# B&R Automation Studio project TD52 (part 79)

#### fPCGVmon.c
```c
/********************************************************************
 * COPYRIGHT -- B&R Industrial Automation GmbH
 ********************************************************************
 * Program: PCGVmon
 * File: fPCGVmon.c
 * Author: 105055527
 * Last modified by: schmisi00
 * Created: Mon Sep 05 18:14:57 2016
 * Last modified: Thu Nov 26 09:45:08 2020
 * Model Version: 0.03
 * Description: Pre-chamber gas valve monitoring (sticking detection).

   Outstandings:
   -------------
   - NA
 * modified Comment: V0.01    22.09.2020    Schmidt,   created initial model
   V0.02    15.10.2020    Schmidt,   modifications after code review / unit testing
   V0.03    26.11.2020    Schmidt,   perm's for class borders (no-hardcoded borders)
 ********************************************************************
 * Implementation of program PCGVmon
 ********************************************************************
 * Generated with B&R Automation Studio Target for Simulink V6.2.0
 * (ERT based)
 ********************************************************************/

#include <bur/plctypes.h>
#include "PCGVmon.h"
#include "rtwtypes.h"

/* Defines */
#define SS_TERMINATE 4
#define SS_OUTPUT 3
#define SS_INITIALIZE 2

/*  Data Types */

/**************************** GLOBAL DATA *************************************/
/*  Definitions */

/*  Declarations  */

/***************************** FILE SCOPE DATA ********************************/

/*************************** FUNCTIONS ****************************************/
#ifdef __cplusplus

unsigned long bur_heap_size = 6553500;

#endif

/*LEGACYMODE_VARIABLES*/
void fPCGVmon(struct fPCGVmon* inst)
{
  tag_RTM_PCGVmon* const PCGVmon_M = &(inst)->bur_PCGVmon;
	inst->bur_PCGVmon.blockIO = &(inst)->bur_BlockIO_PCGVmon;
	inst->bur_PCGVmon.inputs = &(inst)->bur_ExternalInputs_PCGVmon;
	inst->bur_PCGVmon.outputs = &(inst)->bur_ExternalOutputs_PCGVmon;
	inst->bur_PCGVmon.dwork = &(inst)->bur_D_Work_PCGVmon;

  switch (inst->ssMethodType)
  {
   case SS_INITIALIZE:
    /* call model initialize function */
    PCGVmon_initialize(PCGVmon_M, inst);
    break;

   case SS_OUTPUT:
    /* call model step function */
    PCGVmon_step(PCGVmon_M, inst);

    break;

   case SS_TERMINATE:
    /* call model terminate function */
    PCGVmon_terminate(PCGVmon_M, inst);
    break;
  }
}

/*****************************************************************************
   Function block sample time: 1.0s
 *****************************************************************************/

/*****************************************************************************
   B&R Automation Studio Target for Simulink Version: A6.2.0 (28-May-2020)
 *****************************************************************************/

/*======================== TOOL VERSION INFORMATION ==========================*
 * MATLAB 9.8 (R2020a)18-Nov-2019                                             *
 * Simulink 10.1 (R2020a)18-Nov-2019                                          *
 * Simulink Coder 9.3 (R2020a)18-Nov-2019                                     *
 * Embedded Coder 7.4 (R2020a)18-Nov-2019                                     *
 * Stateflow 10.2 (R2020a)18-Nov-2019                                         *
 *============================================================================*/

/*======================= LICENSE IN USE INFORMATION =========================*
 * matlab                                                                     *
 * matlab_coder                                                               *
 * real-time_workshop                                                         *
 * rtw_embedded_coder                                                         *
 * simulink                                                                   *
 *============================================================================*/
```

#### lPCGVmon.fun
```iecst
FUNCTION_BLOCK fPCGVmon
  VAR_INPUT
    ssMethodType: SINT;
  END_VAR
  VAR_INPUT
        Input : tPCGVmon_IN; (*PCGV monitoring bus inputs*)
  END_VAR
  VAR_INPUT
        Perm : tPCGVmon_PERM; (*PCGV monitoring bus perms*)
  END_VAR
  VAR_OUTPUT
        Debug : tPCGVmon_DBG; (*PCGV monitoring bus debug*)
  END_VAR
  VAR_OUTPUT
        Output : tPCGVmon_OUT; (*PCGV monitoring bus outputs*)
  END_VAR
  VAR_OUTPUT
        Version : UDINT; (**)
  END_VAR
	VAR
		bur_BlockIO_PCGVmon : BlockIO_PCGVmon;
	END_VAR
	VAR
		bur_ExternalInputs_PCGVmon : ExternalInputs_PCGVmon;
	END_VAR
	VAR
		bur_ExternalOutputs_PCGVmon : ExternalOutputs_PCGVmon;
	END_VAR
	VAR
		bur_D_Work_PCGVmon : D_Work_PCGVmon;
	END_VAR
	VAR
		bur_PCGVmon : tag_RTM_PCGVmon;
	END_VAR
END_FUNCTION_BLOCK
```

#### lPCGVmon.typ
```iecst
TYPE
	tPCGVmon_DBG :  STRUCT
		bPCGVstick :  ARRAY[0..24] OF BOOL; (*PCGVstickingevent(-)*)
		rTexh_median_diff_grad :  ARRAY[0..24] OF REAL; (**)
		rStdDev :  REAL; (**)
		detectionLim :  REAL; (**)
		rTexh_median_filt :  REAL; (**)
		rU_Ign_Act_Filt :  ARRAY[0..24] OF REAL; (**)
		rTexhMedDeviat :  ARRAY[0..24] OF REAL; (**)
		count1_stick :  ARRAY[0..24] OF REAL; (**)
		count2_stickLong :  ARRAY[0..24] OF REAL; (**)
		unstickDet :  ARRAY[0..24] OF REAL; (**)
		multStickDur :  ARRAY[0..24] OF REAL; (**)
		tiStickDurAll :  ARRAY[0..24] OF REAL; (**)
		bPCGVstickALL :  ARRAY[0..24] OF BOOL; (*PCGVstickingevent(-)*)
		bTexhInRange_out :  ARRAY[0..24] OF BOOL; (*EGTwithinlimit/range(-)*)
	END_STRUCT;

	tPCGVmon_IN :  STRUCT
		rU_Ign_Act :  ARRAY[0..24] OF REAL; (*Actualcylinderignitionvoltage(kV)*)
		MSAGT :  ARRAY[0..24] OF BOOL; (*Cylinderexhaustgastemperaturesensorfailure(-)*)
		rT_EPU_EG :  ARRAY[0..24] OF REAL; (*Cylinderexhaustgastemperature(°C)*)
		tGCB_On_Di :  BOOL; (*Generatorcircuitbreakerclosed(-)*)
		ucNumCyl :  USINT; (*Totalnumberofcylinders(-)*)
		iCnt_PCGV_class1_MM2VIS :  ARRAY[0..24] OF UINT; (*Permclass1counter(MM2VIS)*)
		iCnt_PCGV_class2_MM2VIS :  ARRAY[0..24] OF UINT; (*Permclass2counter(MM2VIS)*)
		iCnt_PCGV_class3_MM2VIS :  ARRAY[0..24] OF UINT; (*Permclass3counter(MM2VIS)*)
		iCnt_PCGV_class4_MM2VIS :  ARRAY[0..24] OF UINT; (*Permclass4counter(MM2VIS)*)
	END_STRUCT;

	tPCGVmon_OUT :  STRUCT
		iCnt_PCGV_class1 :  ARRAY[0..24] OF UINT; (*Class1counter:stickingduration1-10s*)
		iCnt_PCGV_class2 :  ARRAY[0..24] OF UINT; (*Class2counter:stickingduration10-60s*)
		iCnt_PCGV_class3 :  ARRAY[0..24] OF UINT; (*Class3counter:stickingduration60-300s*)
		iCnt_PCGV_class4 :  ARRAY[0..24] OF UINT; (*Class3counter:stickingduration300-3600s*)
		rTi_PCGV_LastStickDur :  REAL; (*Laststickingduration(s)*)
		rTi_PCGV_MeanLastStickEvts :  REAL; (*Stickingdurationoflaststickingevents(s)*)
	END_STRUCT;

	tPCGVmon_PERM :  STRUCT
		bPCGVmon_Act :  BOOL; (*ActivationofPCGVmonitoringandclasscoutnerreset(-)*)
		rU_Ign_DetLim :  REAL; (*MaximumignitionvoltagedroptostillconsiderEGTtemperaturedropasPCGVsticking(kV)*)
		rU_Ign_CylActThresh :  REAL; (*CylinderEGTbelowthisparametertimesignitionvoltagemedianexcludedfrommonitoring(-)*)
		rT_recoverLim :  REAL; (*CylinderEGTrecoverthreshold(°C)*)
		rTi_Uign_MonActDelay :  REAL; (*Activationdelayforignitionvoltageconsiderationinmonitoringfunction(s)*)
		rTmedian_StartThresh :  REAL; (*EGT(median)tobereachedforactivationofignitionvoltageconsideration(°C)*)
		rTi_GCBon_Delay :  REAL; (*ActivationdelayafterGCBclosed(s)*)
		rTi_EGT_ss_ActDelay :  REAL; (*ActivationdelayafterEGTissteadystate(s)*)
		rOffset_EGTgradient_trans :  REAL; (*EGTgradientdetectionlimitoffsetfortransients(-)*)
		rOffset_EGTgradient_ss :  REAL; (*EGTgradientdetectionlimitoffsetforsteadystate(-)*)
		rGradient_LimSwitch :  REAL; (*Switchdetectionlimit(-)*)
		iCnt_PCGV_class1 :  ARRAY[0..24] OF UINT; (*Permclass1counter:stickingduration1-10s*)
		iCnt_PCGV_class2 :  ARRAY[0..24] OF UINT; (*Permclass2counter:stickingduration10-60s*)
		iCnt_PCGV_class3 :  ARRAY[0..24] OF UINT; (*Permclass3counter:stickingduration60-300s*)
		iCnt_PCGV_class4 :  ARRAY[0..24] OF UINT; (*Permclass4counter:stickingduration300-3600s*)
		iTi_PCGV_class1_border :  UINT; (*Permclass1border*)
		iTi_PCGV_class2_border :  UINT; (*Permclass2border*)
		iTi_PCGV_class3_border :  UINT; (*Permclass3border*)
		iTi_PCGV_class4_border :  UINT; (*Permclass4border*)
	END_STRUCT;

END_TYPE

TYPE
rtB_setZero_PCGVmon : STRUCT
	y : ARRAY[0..24] OF REAL;
END_STRUCT;
rtB_TON_PCGVmon : STRUCT
	LogicalOperator3 : BOOL;
END_STRUCT;
rtDW_TON_PCGVmon : STRUCT
	DiscreteTimeIntegrator_DSTATE : REAL;
	DiscreteTimeIntegrator_PrevRese : SINT;
END_STRUCT;
rtB_MATLABFunction_PCGVmon : STRUCT
	y : REAL;
END_STRUCT;
BlockIO_PCGVmon : STRUCT
	BusConversion_InsertedFor_BusOu : tPCGVmon_DBG;
	BusInput : tPCGVmon_IN;
	BusInput1 : tPCGVmon_PERM;
	BusConversion_InsertedFor_Bus_d : tPCGVmon_OUT;
	UnitDelay : UDINT;
	sf_MATLABFunction9 : rtB_MATLABFunction_PCGVmon;
	sf_MATLABFunction8 : rtB_MATLABFunction_PCGVmon;
	sf_MATLABFunction7 : rtB_MATLABFunction_PCGVmon;
	sf_MATLABFunction6 : rtB_MATLABFunction_PCGVmon;
	sf_MATLABFunction5 : rtB_MATLABFunction_PCGVmon;
	sf_MATLABFunction4 : rtB_MATLABFunction_PCGVmon;
	sf_MATLABFunction3_o : rtB_MATLABFunction_PCGVmon;
	sf_MATLABFunction2_o : rtB_MATLABFunction_PCGVmon;
	sf_MATLABFunction10 : rtB_MATLABFunction_PCGVmon;
	sf_MATLABFunction1_p : rtB_MATLABFunction_PCGVmon;
	sf_MATLABFunction : rtB_MATLABFunction_PCGVmon;
	sf_setZero_m : rtB_setZero_PCGVmon;
	TON2 : rtB_TON_PCGVmon;
	TON1 : rtB_TON_PCGVmon;
	TON : rtB_TON_PCGVmon;
	sf_setZero1 : rtB_setZero_PCGVmon;
	sf_setZero : rtB_setZero_PCGVmon;
END_STRUCT;
D_Work_PCGVmon : STRUCT
	Delay_DSTATE : ARRAY[0..74] OF REAL;
	Delay1_DSTATE : ARRAY[0..24] OF REAL;
	UnitDelay2_DSTATE : ARRAY[0..24] OF REAL;
	DelayInput1_DSTATE : REAL;
	UnitDelay13_DSTATE : REAL;
	UnitDelay3_DSTATE : REAL;
	UnitDelay4_DSTATE : REAL;
	UnitDelay5_DSTATE : REAL;
	UnitDelay6_DSTATE : REAL;
	UnitDelay7_DSTATE : REAL;
	UnitDelay8_DSTATE : REAL;
	UnitDelay9_DSTATE : REAL;
	UnitDelay10_DSTATE : REAL;
	UnitDelay11_DSTATE : REAL;
	UnitDelay12_DSTATE : REAL;
	DiscreteTimeIntegrator_DSTATE : REAL;
	DiscreteTimeIntegrator_DSTATE_d : ARRAY[0..24] OF REAL;
	DiscreteTimeIntegrator_DSTATE_b : REAL;
	DiscreteTimeIntegrator_DSTATE_m : ARRAY[0..24] OF REAL;
	UnitDelay_DSTATE : UDINT;
	PrevY : REAL;
	PrevY_a : REAL;
	Cnt1OldDely : ARRAY[0..24] OF REAL;
	Cnt2Old : ARRAY[0..24] OF REAL;
	lastStickDurTmp : ARRAY[0..24] OF REAL;
	count1 : ARRAY[0..24] OF REAL;
	count2 : ARRAY[0..24] OF REAL;
	tiStickDur : ARRAY[0..24] OF REAL;
	tiMultStick : ARRAY[0..24] OF REAL;
	tiStickDurAll : ARRAY[0..24] OF REAL;
	count1Old : ARRAY[0..24] OF REAL;
	iCnt_class1 : ARRAY[0..24] OF UINT;
	iCnt_class2 : ARRAY[0..24] OF UINT;
	iCnt_class3 : ARRAY[0..24] OF UINT;
	iCnt_class4 : ARRAY[0..24] OF UINT;
	iCnt_class1Old : ARRAY[0..24] OF UINT;
	iCnt_class2Old : ARRAY[0..24] OF UINT;
	iCnt_class3Old : ARRAY[0..24] OF UINT;
	iCnt_class4Old : ARRAY[0..24] OF UINT;
	DiscreteTimeIntegrator_PrevRese : SINT;
	DiscreteTimeIntegrator_PrevRe_a : SINT;
	DiscreteTimeIntegrator_PrevRe_p : SINT;
	DiscreteTimeIntegrator_PrevRe_l : SINT;
	DiscreteTimeIntegrator_IC_LOADI : USINT;
	DiscreteTimeIntegrator_IC_LOA_b : USINT;
	DiscreteTimeIntegrator_IC_LOA_l : USINT;
	DiscreteTimeIntegrator_IC_LOA_o : USINT;
	Relay1_Mode : ARRAY[0..24] OF BOOL;
	bPCGVstickTexhGradOld : ARRAY[0..24] OF BOOL;
	bPCGVstick_temp : ARRAY[0..24] OF BOOL;
	bPCGVstickOld : ARRAY[0..24] OF BOOL;
	switch1 : ARRAY[0..24] OF BOOL;
	switch2 : ARRAY[0..24] OF BOOL;
	switch3 : ARRAY[0..24] OF BOOL;
	bTexhInRangeOld : ARRAY[0..24] OF BOOL;
	bTexhInRange : ARRAY[0..24] OF BOOL;
	GCBold : BOOL;
	TON2 : rtDW_TON_PCGVmon;
	TON1 : rtDW_TON_PCGVmon;
	TON : rtDW_TON_PCGVmon;
END_STRUCT;
ExternalInputs_PCGVmon : STRUCT
	In : tPCGVmon_IN;
	Perm : tPCGVmon_PERM;
END_STRUCT;
ExternalOutputs_PCGVmon : STRUCT
	Out : tPCGVmon_OUT;
	Dbg : tPCGVmon_DBG;
END_STRUCT;
tag_RTM_PCGVmon : STRUCT
	errorStatus : REFERENCE TO USINT;
	blockIO : REFERENCE TO BlockIO_PCGVmon;
	inputs : REFERENCE TO ExternalInputs_PCGVmon;
	outputs : REFERENCE TO ExternalOutputs_PCGVmon;
	dwork : REFERENCE TO D_Work_PCGVmon;
END_STRUCT;
emxArray_int32_T_25_PCGVmon : emxArray_int32_T_25;

RT_MODEL_PCGVmon : tag_RTM_PCGVmon;

END_TYPE
TYPE
emxArray_int32_T_25 : STRUCT
	data : ARRAY[0..24] OF DINT;
	size : DINT;
END_STRUCT;
END_TYPE
```

#### lib_properties.txt
```
For manual assignment to hardware configuration please
add the following additional include directories:

\Logical\MATLAB_includes\R2020a\

And the following additional build options:

-lm -D MODEL=PCGVmon -D NUMST=1 -D NCSTATES=0 -D HAVESTDIO -D MODEL_HAS_DYNAMICALLY_LOADED_SFCNS=0 -D CLASSIC_INTERFACE=0 -D ALLOCATIONFCN=0 -D TID01EQ=0 -D TERMFCN=1 -D ONESTEPFCN=1 -D MAT_FILE=0 -D MULTI_INSTANCE_CODE=1 -D INTEGER_CODE=0 -D MT=0
```

#### rt_defines.h
```c
/********************************************************************
 * COPYRIGHT -- B&R Industrial Automation GmbH
 ********************************************************************
 * Program: PCGVmon
 * File: rt_defines.h
 * Author: 105055527
 * Last modified by: schmisi00
 * Created: Mon Sep 05 18:14:57 2016
 * Last modified: Thu Nov 26 09:45:08 2020
 * Model Version: 0.03
 * Description: Pre-chamber gas valve monitoring (sticking detection).

   Outstandings:
   -------------
   - NA
 * modified Comment: V0.01    22.09.2020    Schmidt,   created initial model
   V0.02    15.10.2020    Schmidt,   modifications after code review / unit testing
   V0.03    26.11.2020    Schmidt,   perm's for class borders (no-hardcoded borders)
 ********************************************************************
 * Header for program PCGVmon
 ********************************************************************
 * Generated with B&R Automation Studio Target for Simulink V6.2.0
 * (ERT based)
 ********************************************************************/

#ifndef RTW_HEADER_rt_defines_h_
#define RTW_HEADER_rt_defines_h_
#ifndef MIN
#define MIN(a,b)                       ((a) < (b) ? (a) : (b))
#endif

#ifndef MAX
#define MAX(a,b)                       ((a) > (b) ? (a) : (b))
#endif

#ifndef AST_ROUND
#define AST_ROUND(x)                   ((x)>=0?(long long)((x)+0.5):(long long)((x)-0.5))
#endif

/*===========*
 * Constants *
 *===========*/
#define RT_PI                          3.14159265358979323846
#define RT_PIF                         3.1415927F
#define RT_LN_10                       2.30258509299404568402
#define RT_LN_10F                      2.3025851F
#define RT_LOG10E                      0.43429448190325182765
#define RT_LOG10EF                     0.43429449F
#define RT_E                           2.7182818284590452354
#define RT_EF                          2.7182817F

/*
 * UNUSED_PARAMETER(x)
 *   Used to specify that a function parameter (argument) is required but not
 *   accessed by the function body.
 */
#ifndef UNUSED_PARAMETER
# if defined(__LCC__)
#   define UNUSED_PARAMETER(x)                                   /* do nothing */
# else

/*
 * This is the semi-ANSI standard way of indicating that an
 * unused function parameter is required.
 */
#   define UNUSED_PARAMETER(x)         (void) (x)
# endif
#endif
#endif                                 /* RTW_HEADER_rt_defines_h_ */
```

#### rtwtypes.h
```c
/********************************************************************
 * COPYRIGHT -- B&R Industrial Automation GmbH
 ********************************************************************
 * Program: PCGVmon
 * File: rtwtypes.h
 * Author: 105055527
 * Last modified by: schmisi00
 * Created: Mon Sep 05 18:14:57 2016
 * Last modified: Thu Nov 26 09:45:08 2020
 * Model Version: 0.03
 * Description: Pre-chamber gas valve monitoring (sticking detection).

   Outstandings:
   -------------
   - NA
 * modified Comment: V0.01    22.09.2020    Schmidt,   created initial model
   V0.02    15.10.2020    Schmidt,   modifications after code review / unit testing
   V0.03    26.11.2020    Schmidt,   perm's for class borders (no-hardcoded borders)
 ********************************************************************
 * Header for program PCGVmon
 ********************************************************************
 * Generated with B&R Automation Studio Target for Simulink V6.2.0
 * (ERT based)
 ********************************************************************/

#ifndef RTWTYPES_H
#define RTWTYPES_H

/* Logical type definitions */
#if (!defined(__cplusplus))
#  ifndef false
#   define false                       (0U)
#  endif

#  ifndef true
#   define true                        (1U)
#  endif
#endif

/*=======================================================================*
 * Target hardware information
 *   Device type: Intel->x86/Pentium
 *   Number of bits:     char:   8    short:   16    long:  32
 *                       long:  32
 *                       native word size:  32
 *   Byte ordering: LittleEndian
 *   Signed integer division rounds to: Zero
 *   Shift right on a signed integer as arithmetic shift: on
 *=======================================================================*/

/*=======================================================================*
 * Fixed width word size data types:                                     *
 *   int8_T, int16_T, int32_T     - signed 8, 16, or 32 bit integers     *
 *   uint8_T, uint16_T, uint32_T  - unsigned 8, 16, or 32 bit integers   *
 *   real32_T, real64_T           - 32 and 64 bit floating point numbers *
 *=======================================================================*/
typedef signed char int8_T;
typedef unsigned char uint8_T;
typedef short int16_T;
typedef unsigned short uint16_T;
typedef long int32_T;
typedef unsigned long uint32_T;
typedef float real32_T;
typedef double real64_T;

/*===========================================================================*
 * Generic type definitions: boolean_T, char_T, byte_T, int_T, uint_T,       *
 *                           real_T, time_T, ulong_T.                        *
 *===========================================================================*/
typedef double real_T;
typedef double time_T;
typedef unsigned char boolean_T;
typedef long int_T;
typedef unsigned long uint_T;
typedef unsigned long ulong_T;
typedef char char_T;
typedef unsigned char uchar_T;
typedef char_T byte_T;

/*=======================================================================*
 * Min and Max:                                                          *
 *   int8_T, int16_T, int32_T     - signed 8, 16, or 32 bit integers     *
 *   uint8_T, uint16_T, uint32_T  - unsigned 8, 16, or 32 bit integers   *
 *=======================================================================*/
#define MAX_int8_T                     ((int8_T)(127))
#define MIN_int8_T                     ((int8_T)(-128))
#define MAX_uint8_T                    ((uint8_T)(255U))
#define MAX_int16_T                    ((int16_T)(32767))
#define MIN_int16_T                    ((int16_T)(-32768))
#define MAX_uint16_T                   ((uint16_T)(65535U))
#define MAX_int32_T                    ((int32_T)(2147483647))
#define MIN_int32_T                    ((int32_T)(-2147483647-1))
#define MAX_uint32_T                   ((uint32_T)(0xFFFFFFFFU))

/* Block D-Work pointer type */
typedef void * pointer_T;

#endif                                 /* RTWTYPES_H */

#ifndef MIN
#define MIN(a,b)                       ((a) < (b) ? (a) : (b))
#endif

#ifndef MAX
#define MAX(a,b)                       ((a) > (b) ? (a) : (b))
#endif

#ifndef AST_ROUND
#define AST_ROUND(x)                   ((x)>=0?(long long)((x)+0.5):(long long)((x)-0.5))
#endif
```

### Library Logical/EngineController/Lib_EC/lFSyPrM (ANSIC, version 1.00.0)

#### FSyPrM.c
```c
/********************************************************************
 * COPYRIGHT -- B&R Industrial Automation GmbH
 ********************************************************************
 * Program: FSyPrM
 * File: FSyPrM.c
 * Author: 105055527
 * Last modified by: schmisi00
 * Created: Mon Sep 05 18:14:57 2016
 * Last modified: Mon Jan 25 17:32:20 2021
 * Model Version: 0.08
 * Description: Fast synchronization controller for pre-mixed engines.

   Outstandings:
   -------------
   - NA
 * modified Comment: V0.01    30.03.2020    Schmidt,   project/controller carryover from FSync to FSyncPrM
   V0.02    02.04.2020    Schmidt,   cleanup and deletion of functions not used by pre-mixed engines
   V0.03    12.05.2020    Schmidt,   upgrade to MATLAB/SIMULINK R2020a
   V0.04    14.05.2020    Schmidt,   B&R blocks upgrade to AS Target v6.2.0 (officially supports MATLAB 2020a)
   V0.05    03.08.2020    Schmidt,   changed speed reference for function activation from nominal speed (parameter) to bus bar frequency
   added detection for speed exceedance --> switch over to standard idle controller
   V0.06    04.08.2020    Schmidt,   moved function activation from PARA bus to IN bus
   V0.07    17.08.2020    Schmidt,   included modifications after P6 tests
   V0.08    25.01.2021    Schmidt,   use of frequency based speed set-point (rN_Set) only if rF_MMD_BusBar > 0.5*rF_Nom
 ********************************************************************
 * Implementation of program FSyPrM
 ********************************************************************
 * Generated with B&R Automation Studio Target for Simulink V6.3.1
 * (ERT based)
 ********************************************************************/

#include "FSyPrM.h"
#include "FSyPrM_private.h"

/*  Defines */

/*  Data Types */

/**************************** GLOBAL DATA *************************************/
/*  Definitions */

/*  Declarations  */

/***************************** FILE SCOPE DATA ********************************/

/*************************** FUNCTIONS ****************************************/

/* Model step function */
void FSyPrM_step(RT_MODEL_FSyPrM *const FSyPrM_M, struct fFSyPrM* inst)
{
  struct BlockIO_FSyPrM *FSyPrM_B = ((struct BlockIO_FSyPrM *) FSyPrM_M->blockIO);
  struct D_Work_FSyPrM *FSyPrM_DWork = ((struct D_Work_FSyPrM *) FSyPrM_M->dwork);
  ExternalOutputs_FSyPrM *FSyPrM_Y = (ExternalOutputs_FSyPrM *)
    FSyPrM_M->outputs;
  boolean_T bEnabled;
  real32_T rN_err;
  real32_T rAngle_err;
  real32_T S;
  real32_T gk;
  boolean_T Sf1;
  boolean_T Sf2;
  boolean_T Gplus;
  boolean_T Gminus;
  boolean_T Gammaplus;
  boolean_T Gammaminus;
  boolean_T H1;
  boolean_T H3;
  real32_T rtb_Switch1_i;
  real32_T rtb_DiscreteTimeIntegrator_g;
  int8_T rtb_Switch2;
  real_T rtb_Switch1;
  real32_T S_tmp;
  uint32_T tmp;
  real32_T tmp_0;

  /* S-Function (bur_bus_in): '<Root>/Bus Input' */
  FSyPrM_B->BusInput = inst->In;

  /* S-Function (bur_bus_in): '<Root>/Bus Input1' */
  FSyPrM_B->BusInput1 = inst->Para;

  /* S-Function (bur_bus_in): '<Root>/Bus Input2' */
  FSyPrM_B->BusInput2 = inst->Perm;

  /* Switch: '<S9>/Switch1' incorporates:
   *  Product: '<S9>/Divide1'
   *  Switch: '<S2>/Environment Switch'
   *  Switch: '<S3>/Environment Switch'
   *  Switch: '<S4>/Environment Switch'
   */
  if (FSyPrM_B->BusInput2.bF_act_ena) {
    /* Switch: '<S16>/Switch' incorporates:
     *  Abs: '<S16>/Abs'
     *  RelationalOperator: '<S16>/Relational Operator'
     *  Switch: '<S4>/Environment Switch'
     */
    if (1.0F >= (real32_T)fabs(FSyPrM_B->BusInput1.rF_Nom)) {
      gk = 1.0F;
    } else {
      gk = FSyPrM_B->BusInput1.rF_Nom;
    }

    /* End of Switch: '<S16>/Switch' */
    rtb_Switch1_i = FSyPrM_B->BusInput.rF_MMD * FSyPrM_B->BusInput1.rN_EngNom /
      gk;
  } else {
    rtb_Switch1_i = FSyPrM_B->BusInput.rN_Eng;
  }

  /* End of Switch: '<S9>/Switch1' */

  /* Outputs for Atomic SubSystem: '<S1>/Filter' */
  /* DiscreteIntegrator: '<S10>/Discrete-Time Integrator' incorporates:
   *  Switch: '<S2>/Environment Switch'
   */
  if (FSyPrM_DWork->DiscreteTimeIntegrator_IC_LO_dn != 0) {
    FSyPrM_DWork->DiscreteTimeIntegrator_DSTATE_k = rtb_Switch1_i;
  }

  if (FSyPrM_B->BusInput.bReset ||
      (FSyPrM_DWork->DiscreteTimeIntegrator_PrevRe_d != 0)) {
    FSyPrM_DWork->DiscreteTimeIntegrator_DSTATE_k = rtb_Switch1_i;
  }

  rtb_DiscreteTimeIntegrator_g = FSyPrM_DWork->DiscreteTimeIntegrator_DSTATE_k;

  /* Update for DiscreteIntegrator: '<S10>/Discrete-Time Integrator' */
  FSyPrM_DWork->DiscreteTimeIntegrator_IC_LO_dn = 0U;

  /* Switch: '<S12>/Switch' incorporates:
   *  Abs: '<S12>/Abs'
   *  RelationalOperator: '<S12>/Relational Operator'
   *  Switch: '<S3>/Environment Switch'
   */
  if (2.22044605E-16F >= (real32_T)fabs(FSyPrM_B->BusInput2.rTi_Filtn)) {
    gk = 2.22044605E-16F;
  } else {
    gk = FSyPrM_B->BusInput2.rTi_Filtn;
  }

  /* End of Switch: '<S12>/Switch' */

  /* Update for DiscreteIntegrator: '<S10>/Discrete-Time Integrator' incorporates:
   *  Product: '<S10>/Divide4'
   *  Sum: '<S10>/Sum4'
   *  Switch: '<S2>/Environment Switch'
   */
  FSyPrM_DWork->DiscreteTimeIntegrator_DSTATE_k += (rtb_Switch1_i -
    FSyPrM_DWork->DiscreteTimeIntegrator_DSTATE_k) / gk * 0.01F;
  FSyPrM_DWork->DiscreteTimeIntegrator_PrevRe_d = (int8_T)
    FSyPrM_B->BusInput.bReset;

  /* End of Outputs for SubSystem: '<S1>/Filter' */

  /* Outputs for Atomic SubSystem: '<S1>/Filter1' */
  /* DiscreteIntegrator: '<S11>/Discrete-Time Integrator' incorporates:
   *  Switch: '<S2>/Environment Switch'
   */
  if (FSyPrM_DWork->DiscreteTimeIntegrator_IC_LOA_d != 0) {
    FSyPrM_DWork->DiscreteTimeIntegrator_DSTATE_g = rtb_DiscreteTimeIntegrator_g;
  }

  if (FSyPrM_B->BusInput.bReset ||
      (FSyPrM_DWork->DiscreteTimeIntegrator_PrevRe_h != 0)) {
    FSyPrM_DWork->DiscreteTimeIntegrator_DSTATE_g = rtb_DiscreteTimeIntegrator_g;
  }

  /* Product: '<S11>/Divide4' incorporates:
   *  DiscreteIntegrator: '<S11>/Discrete-Time Integrator'
   *  Sum: '<S11>/Sum4'
   */
  rtb_DiscreteTimeIntegrator_g = (rtb_DiscreteTimeIntegrator_g -
    FSyPrM_DWork->DiscreteTimeIntegrator_DSTATE_g) / 0.01F;

  /* Switch: '<S11>/Switch1' incorporates:
   *  Constant: '<S11>/Constant'
   *  Switch: '<S2>/Environment Switch'
   */
  if (FSyPrM_B->BusInput.bReset) {
    rtb_Switch1 = 0.0;
  } else {
    rtb_Switch1 = rtb_DiscreteTimeIntegrator_g;
  }

  /* End of Switch: '<S11>/Switch1' */

  /* Update for DiscreteIntegrator: '<S11>/Discrete-Time Integrator' incorporates:
   *  Switch: '<S2>/Environment Switch'
   */
  FSyPrM_DWork->DiscreteTimeIntegrator_IC_LOA_d = 0U;
  FSyPrM_DWork->DiscreteTimeIntegrator_DSTATE_g += 0.01F *
    rtb_DiscreteTimeIntegrator_g;
  FSyPrM_DWork->DiscreteTimeIntegrator_PrevRe_h = (int8_T)
    FSyPrM_B->BusInput.bReset;

  /* End of Outputs for SubSystem: '<S1>/Filter1' */

  /* Outputs for Atomic SubSystem: '<S9>/Filter' */
  /* DiscreteIntegrator: '<S18>/Discrete-Time Integrator' incorporates:
   *  Switch: '<S2>/Environment Switch'
   *  Switch: '<S4>/Environment Switch'
   */
  if (FSyPrM_DWork->DiscreteTimeIntegrator_IC_LOADI != 0) {
    FSyPrM_DWork->DiscreteTimeIntegrator_DSTATE = FSyPrM_B->BusInput1.rN_EngNom;
  }

  if (FSyPrM_B->BusInput.bReset ||
      (FSyPrM_DWork->DiscreteTimeIntegrator_PrevRese != 0)) {
    FSyPrM_DWork->DiscreteTimeIntegrator_DSTATE = FSyPrM_B->BusInput1.rN_EngNom;
  }

  rtb_DiscreteTimeIntegrator_g = FSyPrM_DWork->DiscreteTimeIntegrator_DSTATE;

  /* Update for DiscreteIntegrator: '<S18>/Discrete-Time Integrator' */
  FSyPrM_DWork->DiscreteTimeIntegrator_IC_LOADI = 0U;

  /* End of Outputs for SubSystem: '<S9>/Filter' */

  /* Switch: '<S17>/Switch' incorporates:
   *  Abs: '<S17>/Abs'
   *  RelationalOperator: '<S17>/Relational Operator'
   *  Switch: '<S4>/Environment Switch'
   */
  if (1.0F >= (real32_T)fabs(FSyPrM_B->BusInput1.rF_Nom)) {
    gk = 1.0F;
  } else {
    gk = FSyPrM_B->BusInput1.rF_Nom;
  }

  /* End of Switch: '<S17>/Switch' */

  /* Outputs for Atomic SubSystem: '<S9>/Filter' */
  /* Switch: '<S21>/Switch' incorporates:
   *  Abs: '<S21>/Abs'
   *  RelationalOperator: '<S21>/Relational Operator'
   *  Switch: '<S3>/Environment Switch'
   */
  if (2.22044605E-16F >= (real32_T)fabs(FSyPrM_B->BusInput2.rTi_FiltF)) {
    tmp_0 = 2.22044605E-16F;
  } else {
    tmp_0 = FSyPrM_B->BusInput2.rTi_FiltF;
  }

  /* End of Switch: '<S21>/Switch' */

  /* Update for DiscreteIntegrator: '<S18>/Discrete-Time Integrator' incorporates:
   *  Product: '<S18>/Divide4'
   *  Product: '<S9>/Divide'
   *  Sum: '<S18>/Sum4'
   *  Switch: '<S2>/Environment Switch'
   *  Switch: '<S4>/Environment Switch'
   */
  FSyPrM_DWork->DiscreteTimeIntegrator_DSTATE +=
    (FSyPrM_B->BusInput.rF_MMD_BusBar / gk * FSyPrM_B->BusInput1.rN_EngNom -
     FSyPrM_DWork->DiscreteTimeIntegrator_DSTATE) / tmp_0 * 0.01F;
  FSyPrM_DWork->DiscreteTimeIntegrator_PrevRese = (int8_T)
    FSyPrM_B->BusInput.bReset;

  /* End of Outputs for SubSystem: '<S9>/Filter' */

  /* Switch: '<S9>/Switch' incorporates:
   *  Constant: '<S9>/Constant1'
   *  Logic: '<S9>/Logical Operator'
   *  Product: '<S9>/Product'
   *  RelationalOperator: '<S9>/Relational Operator'
   *  Switch: '<S2>/Environment Switch'
   *  Switch: '<S3>/Environment Switch'
   *  Switch: '<S4>/Environment Switch'
   */
  if (FSyPrM_B->BusInput2.bSpeedSet_ena || (FSyPrM_B->BusInput.rF_MMD_BusBar <
       0.5F * FSyPrM_B->BusInput1.rF_Nom)) {
    rtb_DiscreteTimeIntegrator_g = FSyPrM_B->BusInput1.rN_EngNom;
  }

  /* End of Switch: '<S9>/Switch' */

  /* MATLAB Function: '<Root>/Skipfire_active' incorporates:
   *  Switch: '<S2>/Environment Switch'
   *  Switch: '<S3>/Environment Switch'
   */
  /* MATLAB Function 'Skipfire_active': '<S7>:1' */
  if (FSyPrM_B->BusInput.rN_Eng >= FSyPrM_B->BusInput2.rN_enableNorm *
      rtb_DiscreteTimeIntegrator_g) {
    /* '<S7>:1:16' */
    /* '<S7>:1:17' */
    FSyPrM_DWork->ssr = true;
  }

  if ((rtb_Switch1 < FSyPrM_B->BusInput2.rN_dot_release) && ((real32_T)fabs
       (FSyPrM_B->BusInput.rN_Eng - rtb_DiscreteTimeIntegrator_g) <
       FSyPrM_B->BusInput2.rN_SpdSettled)) {
    /* '<S7>:1:20' */
    /* '<S7>:1:21' */
    FSyPrM_DWork->spd_settled = true;
  }

  if (FSyPrM_DWork->spd_settled && ((real32_T)fabs(FSyPrM_B->BusInput.rN_Eng -
        rtb_DiscreteTimeIntegrator_g) > FSyPrM_B->BusInput2.rN_SpdDevMax)) {
    /* '<S7>:1:24' */
    /* '<S7>:1:25' */
    FSyPrM_DWork->spd_DevExc = true;
  }

  if (FSyPrM_B->BusInput.bGCB_ON || (FSyPrM_B->BusInput.rN_Eng < 100.0F)) {
    /* '<S7>:1:28' */
    /* '<S7>:1:29' */
    FSyPrM_DWork->ssr = false;

    /* '<S7>:1:30' */
    FSyPrM_DWork->spd_settled = false;

    /* '<S7>:1:31' */
    FSyPrM_DWork->spd_DevExc = false;
  }

  /* Switch: '<S9>/Switch2' incorporates:
   *  Constant: '<S9>/Constant'
   *  Switch: '<S2>/Environment Switch'
   *  Switch: '<S3>/Environment Switch'
   */
  /* '<S7>:1:35' */
  /* '<S7>:1:36' */
  /* '<S7>:1:37' */
  if (FSyPrM_B->BusInput.bFastSync) {
    rtb_Switch2 = FSyPrM_B->BusInput2.iCtrSel;
  } else {
    rtb_Switch2 = 0;
  }

  /* End of Switch: '<S9>/Switch2' */

  /* MATLAB Function: '<Root>/FSyncITPCtrl' incorporates:
   *  Gain: '<S9>/Conv rad'
   *  MATLAB Function: '<Root>/Skipfire_active'
   *  Outport: '<Root>/dbg'
   *  Product: '<S8>/Product1'
   *  SampleTimeMath: '<S8>/Weighted Sample Time'
   *  Switch: '<S2>/Environment Switch'
   *  Switch: '<S3>/Environment Switch'
   *
   * About '<S8>/Weighted Sample Time':
   *  y = K where K = 1 / ( w * Ts )
   */
  /* MATLAB Function 'FSyncITPCtrl': '<S5>:1' */
  if ((!FSyPrM_DWork->CA_retarded_not_empty) || (!FSyPrM_DWork->ssr) ||
      (rtb_Switch2 == 0)) {
    /* '<S5>:1:10' */
    /* '<S5>:1:11' */
    FSyPrM_DWork->CA_retarded = FSyPrM_B->BusInput2.rCA_ITPRetardMax;
    FSyPrM_DWork->CA_retarded_not_empty = true;

    /* '<S5>:1:12' */
    FSyPrM_DWork->retardcounter = 0U;

    /* '<S5>:1:13' */
    FSyPrM_DWork->Count_Switch = 0U;
  }

  if (FSyPrM_DWork->spd_settled) {
    /* '<S5>:1:18' */
    if ((FSyPrM_DWork->Count_Switch < FSyPrM_B->BusInput2.rTi_FastSync * 100.0F)
        && (rtb_Switch2 >= 1) && (!FSyPrM_DWork->spd_DevExc)) {
      /* '<S5>:1:19' */
      /* '<S5>:1:20' */
      tmp = FSyPrM_DWork->Count_Switch + 1U;
      if (tmp > 65535U) {
        tmp = 65535U;
      }

      FSyPrM_DWork->Count_Switch = (uint16_T)tmp;

      /* '<S5>:1:21' */
      bEnabled = true;
    } else {
      /* '<S5>:1:23' */
      bEnabled = false;
    }
  } else {
    /* '<S5>:1:26' */
    bEnabled = false;
  }

  if (FSyPrM_DWork->retardcounter < 2000) {
    /* '<S5>:1:30' */
    /* '<S5>:1:31' */
    tmp = FSyPrM_DWork->retardcounter + 1U;
    if (tmp > 65535U) {
      tmp = 65535U;
    }

    FSyPrM_DWork->retardcounter = (uint16_T)tmp;
  } else {
    /* '<S5>:1:33' */
    FSyPrM_DWork->retardcounter = 0U;
  }

  /* '<S5>:1:39' */
  rN_err = rtb_Switch1_i - rtb_DiscreteTimeIntegrator_g;

  /* '<S5>:1:40' */
  rAngle_err = 0.0174532924F * FSyPrM_B->BusInput.rAng_MMD_Diff -
    FSyPrM_B->BusInput2.rAngleSetDeg * 3.14159274F / 180.0F;

  /* '<S5>:1:42' */
  S_tmp = (real32_T)fabs(rN_err);
  S = 0.5F * rN_err * S_tmp * 2.0F * 3.14159274F / 30.0F * 2.0F * 3.14159274F /
    30.0F + rAngle_err;
  if ((0.5F * rN_err * rN_err * 2.0F * 3.14159274F / 30.0F * 2.0F * 3.14159274F /
       30.0F + rAngle_err == 0.0F) && (rN_err >= 0.0F)) {
    /* '<S5>:1:43' */
    Sf1 = true;
  } else {
    Sf1 = false;
  }

  gk = -0.5F * rN_err * rN_err * 2.0F * 3.14159274F / 30.0F * 2.0F * 3.14159274F
    / 30.0F + rAngle_err;
  if ((gk == 0.0F) && (rN_err <= 0.0F)) {
    /* '<S5>:1:44' */
    Sf2 = true;
  } else {
    Sf2 = false;
  }

  /* '<S5>:1:45' */
  tmp_0 = FSyPrM_B->BusInput2.rRelaxAngleDeg * 3.14159274F / 180.0F;
  if ((S <= tmp_0) && (S >= -FSyPrM_B->BusInput2.rRelaxAngleDeg * 3.14159274F /
                       180.0F) && (-rN_err < 0.0F)) {
    /* '<S5>:1:47' */
    Gplus = true;
  } else {
    Gplus = false;
  }

  if ((S <= tmp_0) && (S >= -FSyPrM_B->BusInput2.rRelaxAngleDeg * 3.14159274F /
                       180.0F) && (-rN_err > 0.0F)) {
    /* '<S5>:1:48' */
    Gminus = true;
  } else {
    Gminus = false;
  }

  /* '<S5>:1:49' */
  /* '<S5>:1:50' */
  /* '<S5>:1:51' */
  if ((gk == tmp_0) && (-rN_err < 0.0F)) {
    /* '<S5>:1:52' */
    Gammaplus = true;
  } else {
    Gammaplus = false;
  }

  gk = -FSyPrM_B->BusInput2.rRelaxAngleDeg * 3.14159274F / 180.0F;
  if ((gk == S) && (-rN_err > 0.0F)) {
    /* '<S5>:1:53' */
    Gammaminus = true;
  } else {
    Gammaminus = false;
  }

  if (Gplus || (S < gk)) {
    /* '<S5>:1:54' */
    Gplus = true;
  }

  if (Gminus || (S > tmp_0)) {
    /* '<S5>:1:55' */
    Gminus = true;
  }

  /* '<S5>:1:57' */
  gk = (FSyPrM_B->BusInput2.rWeightFuel + 4.0F) / (2.0F *
    FSyPrM_B->BusInput2.rWeightFuel);
  if ((S >= 0.0F) && (gk * rN_err * S_tmp * 2.0F * 3.14159274F / 30.0F * 2.0F *
                      3.14159274F / 30.0F + rAngle_err > 0.0F)) {
    /* '<S5>:1:58' */
    H1 = true;
  } else {
    H1 = false;
  }

  if ((S <= 0.0F) && (gk * rN_err * (real32_T)fabs(rN_err) * 2.0F * 3.14159274F /
                      30.0F * 2.0F * 3.14159274F / 30.0F + rAngle_err < 0.0F)) {
    /* '<S5>:1:60' */
    H3 = true;
  } else {
    H3 = false;
  }

  if ((S > 0.0F) && (gk * rN_err * (real32_T)fabs(rN_err) * 2.0F * 3.14159274F /
                     30.0F * 2.0F * 3.14159274F / 30.0F + rAngle_err <= 0.0F)) {
    /* '<S5>:1:61' */
    FSyPrM_Y->dbg.H4 = true;
  } else {
    FSyPrM_Y->dbg.H4 = false;
  }

  /* '<S5>:1:62' */
  /* '<S5>:1:66' */
  switch (rtb_Switch2) {
   case 1:
    if ((S > FSyPrM_B->BusInput2.rHystOptimal) || (Sf2 && FSyPrM_DWork->ssr)) {
      /* '<S5>:1:68' */
      /* '<S5>:1:69' */
      FSyPrM_DWork->CA_retarded = FSyPrM_B->BusInput2.rCA_ITPRetardMin;

      /* '<S5>:1:70' */
      FSyPrM_DWork->retardcounter = 0U;
    } else {
      if ((S < -FSyPrM_B->BusInput2.rHystOptimal) || (Sf1 && FSyPrM_DWork->ssr))
      {
        /* '<S5>:1:71' */
        /* '<S5>:1:72' */
        FSyPrM_DWork->CA_retarded = FSyPrM_B->BusInput2.rCA_ITPRetardMax;

        /* '<S5>:1:73' */
        FSyPrM_DWork->retardcounter = 0U;
      }
    }
    break;

   case 2:
    if ((Gminus || Gammaminus) && FSyPrM_DWork->ssr) {
      /* '<S5>:1:77' */
      /* '<S5>:1:78' */
      FSyPrM_DWork->CA_retarded = FSyPrM_B->BusInput2.rCA_ITPRetardMin;

      /* '<S5>:1:79' */
      FSyPrM_DWork->retardcounter = 0U;
    } else {
      if ((Gplus || Gammaplus) && FSyPrM_DWork->ssr) {
        /* '<S5>:1:80' */
        /* '<S5>:1:81' */
        FSyPrM_DWork->CA_retarded = FSyPrM_B->BusInput2.rCA_ITPRetardMax;

        /* '<S5>:1:82' */
        FSyPrM_DWork->retardcounter = 0U;
      }
    }
    break;

   case 3:
    if (H1 && FSyPrM_DWork->ssr) {
      /* '<S5>:1:86' */
      /* '<S5>:1:87' */
      FSyPrM_DWork->CA_retarded = FSyPrM_B->BusInput2.rCA_ITPRetardMin;

      /* '<S5>:1:88' */
      FSyPrM_DWork->retardcounter = 0U;
    } else {
      if (H3 && FSyPrM_DWork->ssr) {
        /* '<S5>:1:89' */
        /* '<S5>:1:90' */
        FSyPrM_DWork->CA_retarded = FSyPrM_B->BusInput2.rCA_ITPRetardMax;

        /* '<S5>:1:91' */
        FSyPrM_DWork->retardcounter = 0U;
      }
    }
    break;

   default:
    /* '<S5>:1:99' */
    FSyPrM_DWork->CA_retarded = FSyPrM_B->BusInput2.rCA_ITPRetardMax;

    /* '<S5>:1:100' */
    FSyPrM_DWork->retardcounter = 0U;
    break;
  }

  if (!FSyPrM_DWork->ssr) {
    /* Outport: '<Root>/rRetardITP' */
    /* '<S5>:1:105' */
    /* '<S5>:1:106' */
    FSyPrM_Y->rRetardITP = FSyPrM_B->BusInput2.rCA_ITPRetardMax;
  } else if (bEnabled) {
    /* Outport: '<Root>/rRetardITP' */
    /* '<S5>:1:108' */
    /* '<S5>:1:109' */
    FSyPrM_Y->rRetardITP = FSyPrM_DWork->CA_retarded;
  } else {
    /* Outport: '<Root>/rRetardITP' */
    /* '<S5>:1:111' */
    FSyPrM_Y->rRetardITP = FSyPrM_B->BusInput2.rCA_ITPRetardMax;
  }

  /* '<S5>:1:116' */
  FSyPrM_Y->dbg.iRetardCounter = FSyPrM_DWork->retardcounter;

  /* '<S5>:1:117' */
  FSyPrM_Y->dbg.rSwitchSurf = S;

  /* '<S5>:1:118' */
  FSyPrM_Y->dbg.Sf1 = Sf1;

  /* '<S5>:1:119' */
  FSyPrM_Y->dbg.Sf2 = Sf2;

  /* '<S5>:1:120' */
  FSyPrM_Y->dbg.H3 = H3;

  /* '<S5>:1:121' */
  /* '<S5>:1:122' */
  FSyPrM_Y->dbg.rSmodSlid = 10.0F * rN_err * 2.0F * 3.14159274F / 30.0F * 2.0F *
    3.14159274F / 30.0F + rAngle_err;

  /* '<S5>:1:123' */
  FSyPrM_Y->dbg.iCounterSwitch = FSyPrM_DWork->Count_Switch;

  /* '<S5>:1:124' */
  FSyPrM_Y->dbg.bEna = FSyPrM_DWork->ssr;

  /* '<S5>:1:125' */
  FSyPrM_Y->dbg.iCtrSel = rtb_Switch2;

  /* '<S5>:1:126' */
  FSyPrM_Y->dbg.rN_Set = rtb_DiscreteTimeIntegrator_g;

  /* '<S5>:1:127' */
  FSyPrM_Y->dbg.rN_Eng = rtb_Switch1_i;

  /* '<S5>:1:128' */
  FSyPrM_Y->dbg.bSpdSettled = FSyPrM_DWork->spd_settled;

  /* '<S5>:1:129' */
  FSyPrM_Y->dbg.rN_dot = (real32_T)rtb_Switch1;
  FSyPrM_B->bEnabled = bEnabled;

  /* End of MATLAB Function: '<Root>/FSyncITPCtrl' */

  /* S-Function (bur_bus_out): '<Root>/Bus Output' incorporates:
   *  Outport: '<Root>/dbg'
   */
  inst->Dbg = FSyPrM_Y->dbg;

  /* S-Function (bur_out): '<Root>/Output1' */
  inst->bEnabled = FSyPrM_B->bEnabled;

  /* S-Function (bur_out): '<Root>/Output2' incorporates:
   *  Outport: '<Root>/rRetardITP'
   */
  inst->rRetardITP = FSyPrM_Y->rRetardITP;

  /* UnitDelay: '<S6>/Unit Delay' */
  FSyPrM_B->UnitDelay = FSyPrM_DWork->UnitDelay_DSTATE;

  /* S-Function (bur_out): '<Root>/Output' */
  inst->Version = FSyPrM_B->UnitDelay;

  /* Update for UnitDelay: '<S6>/Unit Delay' */
  FSyPrM_DWork->UnitDelay_DSTATE = 8U;
}

/* Model initialize function */
void FSyPrM_initialize(RT_MODEL_FSyPrM *const FSyPrM_M, struct fFSyPrM* inst)
{
  struct D_Work_FSyPrM *FSyPrM_DWork = ((struct D_Work_FSyPrM *) FSyPrM_M->dwork);

  /* SystemInitialize for Atomic SubSystem: '<S1>/Filter' */
  /* InitializeConditions for DiscreteIntegrator: '<S10>/Discrete-Time Integrator' */
  FSyPrM_DWork->DiscreteTimeIntegrator_IC_LO_dn = 1U;

  /* End of SystemInitialize for SubSystem: '<S1>/Filter' */

  /* SystemInitialize for Atomic SubSystem: '<S1>/Filter1' */
  /* InitializeConditions for DiscreteIntegrator: '<S11>/Discrete-Time Integrator' */
  FSyPrM_DWork->DiscreteTimeIntegrator_IC_LOA_d = 1U;

  /* End of SystemInitialize for SubSystem: '<S1>/Filter1' */

  /* SystemInitialize for Atomic SubSystem: '<S9>/Filter' */
  /* InitializeConditions for DiscreteIntegrator: '<S18>/Discrete-Time Integrator' */
  FSyPrM_DWork->DiscreteTimeIntegrator_IC_LOADI = 1U;

  /* End of SystemInitialize for SubSystem: '<S9>/Filter' */
}

/* Model terminate function */
void FSyPrM_terminate(RT_MODEL_FSyPrM *const FSyPrM_M, struct fFSyPrM* inst)
{
  /* (no terminate code required) */
  UNUSED_PARAMETER(FSyPrM_M);
}

/*======================== TOOL VERSION INFORMATION ==========================*
 * MATLAB 9.8 (R2020a)18-Nov-2019                                             *
 * Simulink 10.1 (R2020a)18-Nov-2019                                          *
 * Simulink Coder 9.3 (R2020a)18-Nov-2019                                     *
 * Embedded Coder 7.4 (R2020a)18-Nov-2019                                     *
 * Stateflow 10.2 (R2020a)18-Nov-2019                                         *
 *============================================================================*/

/*======================= LICENSE IN USE INFORMATION =========================*
 * matlab                                                                     *
 * matlab_coder                                                               *
 * real-time_workshop                                                         *
 * rtw_embedded_coder                                                         *
 * simulink                                                                   *
 *============================================================================*/
```

#### FSyPrM.h
```c
/********************************************************************
 * COPYRIGHT -- B&R Industrial Automation GmbH
 ********************************************************************
 * Program: FSyPrM
 * File: FSyPrM.h
 * Author: 105055527
 * Last modified by: schmisi00
 * Created: Mon Sep 05 18:14:57 2016
 * Last modified: Mon Jan 25 17:32:20 2021
 * Model Version: 0.08
 * Description: Fast synchronization controller for pre-mixed engines.

   Outstandings:
   -------------
   - NA
 * modified Comment: V0.01    30.03.2020    Schmidt,   project/controller carryover from FSync to FSyncPrM
   V0.02    02.04.2020    Schmidt,   cleanup and deletion of functions not used by pre-mixed engines
   V0.03    12.05.2020    Schmidt,   upgrade to MATLAB/SIMULINK R2020a
   V0.04    14.05.2020    Schmidt,   B&R blocks upgrade to AS Target v6.2.0 (officially supports MATLAB 2020a)
   V0.05    03.08.2020    Schmidt,   changed speed reference for function activation from nominal speed (parameter) to bus bar frequency
   added detection for speed exceedance --> switch over to standard idle controller
   V0.06    04.08.2020    Schmidt,   moved function activation from PARA bus to IN bus
   V0.07    17.08.2020    Schmidt,   included modifications after P6 tests
   V0.08    25.01.2021    Schmidt,   use of frequency based speed set-point (rN_Set) only if rF_MMD_BusBar > 0.5*rF_Nom
 ********************************************************************
 * Header for program FSyPrM
 ********************************************************************
 * Generated with B&R Automation Studio Target for Simulink V6.3.1
 * (ERT based)
 ********************************************************************/

#ifndef RTW_HEADER_FSyPrM_h_
#define RTW_HEADER_FSyPrM_h_
#include <math.h>
#ifndef FSyPrM_COMMON_INCLUDES_
# define FSyPrM_COMMON_INCLUDES_
#include "rtwtypes.h"
#endif                                 /* FSyPrM_COMMON_INCLUDES_ */

#include "FSyPrM_types.h"
#include "lFSyPrM.h"
/* Beginning of Dynamic TypeDefs: */
/* End of Dynamic TypeDefs: */
#ifndef MIN
#define MIN(a,b)	((a) < (b) ? (a) : (b))
#endif

#ifndef MAX
#define MAX(a,b)	((a) > (b) ? (a) : (b))
#endif

#ifndef AST_ROUND
#define AST_ROUND(x) ((x)>=0?(long long)((x)+0.5):(long long)((x)-0.5))
#endif

#include "rt_defines.h"

/* Macros for accessing real-time model data structure */
#ifndef rtmGetBlockIO
# define rtmGetBlockIO(rtm)            ((rtm)->blockIO)
#endif

#ifndef rtmSetBlockIO
# define rtmSetBlockIO(rtm, val)       ((rtm)->blockIO = (val))
#endif

#ifndef rtmGetRootDWork
# define rtmGetRootDWork(rtm)          ((rtm)->dwork)
#endif

#ifndef rtmSetRootDWork
# define rtmSetRootDWork(rtm, val)     ((rtm)->dwork = (val))
#endif

#ifndef rtmGetU
# define rtmGetU(rtm)                  ((rtm)->inputs)
#endif

#ifndef rtmSetU
# define rtmSetU(rtm, val)             ((rtm)->inputs = (val))
#endif

#ifndef rtmGetY
# define rtmGetY(rtm)                  ((rtm)->outputs)
#endif

#ifndef rtmSetY
# define rtmSetY(rtm, val)             ((rtm)->outputs = (val))
#endif

#ifndef rtmGetErrorStatus
# define rtmGetErrorStatus(rtm)        ((rtm)->errorStatus)
#endif

#ifndef rtmSetErrorStatus
# define rtmSetErrorStatus(rtm, val)   ((rtm)->errorStatus = (val))
#endif

#ifndef MIN
#define MIN(a,b)                       ((a) < (b) ? (a) : (b))
#endif

#ifndef MAX
#define MAX(a,b)                       ((a) > (b) ? (a) : (b))
#endif

#ifndef AST_ROUND
#define AST_ROUND(x)                   ((x)>=0?(long long)((x)+0.5):(long long)((x)-0.5))
#endif

/* user code (top of header file) */
/***************************************************************************************************
 * COPYRIGHT -- INNIO Jenbacher GmbH & CO OG
 ****************************************************************************************************
 * Program:            FSyPrM
 * Author:             schmisi00
 * Created:            25.01.2021 17:32
 ****************************************************************************************************
 * MODEL INFORMATION
 ****************************************************************************************************
 * Model Name:         C:\Git\FastSync_PreMixed\03_Simulation\FSyPrM.slx
 * Model Version:      0.08
 * Simulink Version:   R2020a
 * B&R Target:         V6.3.1
 * Description:        Fast synchronization controller for pre-mixed engines.
 *
 *                     Outstandings:
 *                     -------------
 *                     - NA
 ****************************************************************************************************
 * HISTORY
 ****************************************************************************************************
 * Last Modified By:   schmisi00
 * Last Modified Date: Mon Jan 25 17:31:53 2021
 * Modified Comment:   V0.01    30.03.2020    Schmidt,   project/controller carryover from FSync to FSyncPrM
 *                     V0.02    02.04.2020    Schmidt,   cleanup and deletion of functions not used by pre-mixed engines
 *                     V0.03    12.05.2020    Schmidt,   upgrade to MATLAB/SIMULINK R2020a
 *                     V0.04    14.05.2020    Schmidt,   B&R blocks upgrade to AS Target v6.2.0 (officially supports MATLAB 2020a)
 *                     V0.05    03.08.2020    Schmidt,   changed speed reference for function activation from nominal speed (parameter) to bus bar frequency
 *                                                                          added detection for speed exceedance --> switch over to standard idle controller
 *                     V0.06    04.08.2020    Schmidt,   moved function activation from PARA bus to IN bus
 *                     V0.07    17.08.2020    Schmidt,   included modifications after P6 tests
 *                     V0.08    25.01.2021    Schmidt,   use of frequency based speed set-point (rN_Set) only if rF_MMD_BusBar > 0.5*rF_Nom
 ****************************************************************************************************/

/* Block signals (default storage) */

/* Block states (default storage) for system '<Root>' */

/* External inputs (root inport signals with default storage) */

/* External outputs (root outports fed by signals with default storage) */

/* Real-time Model Data Structure */

/* Model entry point functions */
extern void FSyPrM_initialize(RT_MODEL_FSyPrM *const FSyPrM_M, struct fFSyPrM* inst);
extern void FSyPrM_step(RT_MODEL_FSyPrM *const FSyPrM_M, struct fFSyPrM* inst);
extern void FSyPrM_terminate(RT_MODEL_FSyPrM *const FSyPrM_M, struct fFSyPrM* inst);

/*-
 * The generated code includes comments that allow you to trace directly
 * back to the appropriate location in the model.  The basic format
 * is <system>/block_name, where system is the system number (uniquely
 * assigned by Simulink) and block_name is the name of the block.
 *
 * Use the MATLAB hilite_system command to trace the generated code back
 * to the model.  For example,
 *
 * hilite_system('<S3>')    - opens system 3
 * hilite_system('<S3>/Kp') - opens and selects block Kp which resides in S3
 *
 * Here is the system hierarchy for this model
 *
 * '<Root>' : 'FSyPrM'
 * '<S1>'   : 'FSyPrM/EngSpeedGradient'
 * '<S2>'   : 'FSyPrM/Environment Controller3'
 * '<S3>'   : 'FSyPrM/Environment Controller4'
 * '<S4>'   : 'FSyPrM/Environment Controller5'
 * '<S5>'   : 'FSyPrM/FSyncITPCtrl'
 * '<S6>'   : 'FSyPrM/Info'
 * '<S7>'   : 'FSyPrM/Skipfire_active'
 * '<S8>'   : 'FSyPrM/Time2Sample'
 * '<S9>'   : 'FSyPrM/ValueSelect'
 * '<S10>'  : 'FSyPrM/EngSpeedGradient/Filter'
 * '<S11>'  : 'FSyPrM/EngSpeedGradient/Filter1'
 * '<S12>'  : 'FSyPrM/EngSpeedGradient/Filter/Divisor'
 * '<S13>'  : 'FSyPrM/EngSpeedGradient/Filter/Divisor/Data Type Conversion Inherited'
 * '<S14>'  : 'FSyPrM/EngSpeedGradient/Filter1/Divisor'
 * '<S15>'  : 'FSyPrM/EngSpeedGradient/Filter1/Divisor/Data Type Conversion Inherited'
 * '<S16>'  : 'FSyPrM/ValueSelect/Divisor'
 * '<S17>'  : 'FSyPrM/ValueSelect/Divisor1'
 * '<S18>'  : 'FSyPrM/ValueSelect/Filter'
 * '<S19>'  : 'FSyPrM/ValueSelect/Divisor/Data Type Conversion Inherited'
 * '<S20>'  : 'FSyPrM/ValueSelect/Divisor1/Data Type Conversion Inherited'
 * '<S21>'  : 'FSyPrM/ValueSelect/Filter/Divisor'
 * '<S22>'  : 'FSyPrM/ValueSelect/Filter/Divisor/Data Type Conversion Inherited'
 */
#endif                                 /* RTW_HEADER_FSyPrM_h_ */
```

#### FSyPrM_private.h
```c
/********************************************************************
 * COPYRIGHT -- B&R Industrial Automation GmbH
 ********************************************************************
 * Program: FSyPrM
 * File: FSyPrM_private.h
 * Author: 105055527
 * Last modified by: schmisi00
 * Created: Mon Sep 05 18:14:57 2016
 * Last modified: Mon Jan 25 17:32:20 2021
 * Model Version: 0.08
 * Description: Fast synchronization controller for pre-mixed engines.

   Outstandings:
   -------------
   - NA
 * modified Comment: V0.01    30.03.2020    Schmidt,   project/controller carryover from FSync to FSyncPrM
   V0.02    02.04.2020    Schmidt,   cleanup and deletion of functions not used by pre-mixed engines
   V0.03    12.05.2020    Schmidt,   upgrade to MATLAB/SIMULINK R2020a
   V0.04    14.05.2020    Schmidt,   B&R blocks upgrade to AS Target v6.2.0 (officially supports MATLAB 2020a)
   V0.05    03.08.2020    Schmidt,   changed speed reference for function activation from nominal speed (parameter) to bus bar frequency
   added detection for speed exceedance --> switch over to standard idle controller
   V0.06    04.08.2020    Schmidt,   moved function activation from PARA bus to IN bus
   V0.07    17.08.2020    Schmidt,   included modifications after P6 tests
   V0.08    25.01.2021    Schmidt,   use of frequency based speed set-point (rN_Set) only if rF_MMD_BusBar > 0.5*rF_Nom
 ********************************************************************
 * Header for program FSyPrM
 ********************************************************************
 * Generated with B&R Automation Studio Target for Simulink V6.3.1
 * (ERT based)
 ********************************************************************/

#ifndef RTW_HEADER_FSyPrM_private_h_
#define RTW_HEADER_FSyPrM_private_h_
#include "rtwtypes.h"
#include <bur/plctypes.h>
#ifndef MIN
#define MIN(a,b)                       ((a) < (b) ? (a) : (b))
#endif

#ifndef MAX
#define MAX(a,b)                       ((a) > (b) ? (a) : (b))
#endif

#ifndef AST_ROUND
#define AST_ROUND(x)                   ((x)>=0?(long long)((x)+0.5):(long long)((x)-0.5))
#endif
#endif                                 /* RTW_HEADER_FSyPrM_private_h_ */
```

#### FSyPrM_types.h
```c
/********************************************************************
 * COPYRIGHT -- B&R Industrial Automation GmbH
 ********************************************************************
 * Program: FSyPrM
 * File: FSyPrM_types.h
 * Author: 105055527
 * Last modified by: schmisi00
 * Created: Mon Sep 05 18:14:57 2016
 * Last modified: Mon Jan 25 17:32:20 2021
 * Model Version: 0.08
 * Description: Fast synchronization controller for pre-mixed engines.

   Outstandings:
   -------------
   - NA
 * modified Comment: V0.01    30.03.2020    Schmidt,   project/controller carryover from FSync to FSyncPrM
   V0.02    02.04.2020    Schmidt,   cleanup and deletion of functions not used by pre-mixed engines
   V0.03    12.05.2020    Schmidt,   upgrade to MATLAB/SIMULINK R2020a
   V0.04    14.05.2020    Schmidt,   B&R blocks upgrade to AS Target v6.2.0 (officially supports MATLAB 2020a)
   V0.05    03.08.2020    Schmidt,   changed speed reference for function activation from nominal speed (parameter) to bus bar frequency
   added detection for speed exceedance --> switch over to standard idle controller
   V0.06    04.08.2020    Schmidt,   moved function activation from PARA bus to IN bus
   V0.07    17.08.2020    Schmidt,   included modifications after P6 tests
   V0.08    25.01.2021    Schmidt,   use of frequency based speed set-point (rN_Set) only if rF_MMD_BusBar > 0.5*rF_Nom
 ********************************************************************
 * Header for program FSyPrM
 ********************************************************************
 * Generated with B&R Automation Studio Target for Simulink V6.3.1
 * (ERT based)
 ********************************************************************/

#ifndef RTW_HEADER_FSyPrM_types_h_
#define RTW_HEADER_FSyPrM_types_h_
#include "rtwtypes.h"

/* Model Code Variants */
#ifndef MIN
#define MIN(a,b)                       ((a) < (b) ? (a) : (b))
#endif

#ifndef MAX
#define MAX(a,b)                       ((a) > (b) ? (a) : (b))
#endif

#ifndef AST_ROUND
#define AST_ROUND(x)                   ((x)>=0?(long long)((x)+0.5):(long long)((x)-0.5))
#endif

/* Forward declaration for rtModel */

#endif                                 /* RTW_HEADER_FSyPrM_types_h_ */
```

#### fFSyPrM.c
```c
/********************************************************************
 * COPYRIGHT -- B&R Industrial Automation GmbH
 ********************************************************************
 * Program: FSyPrM
 * File: fFSyPrM.c
 * Author: 105055527
 * Last modified by: schmisi00
 * Created: Mon Sep 05 18:14:57 2016
 * Last modified: Mon Jan 25 17:32:20 2021
 * Model Version: 0.08
 * Description: Fast synchronization controller for pre-mixed engines.

   Outstandings:
   -------------
   - NA
 * modified Comment: V0.01    30.03.2020    Schmidt,   project/controller carryover from FSync to FSyncPrM
   V0.02    02.04.2020    Schmidt,   cleanup and deletion of functions not used by pre-mixed engines
   V0.03    12.05.2020    Schmidt,   upgrade to MATLAB/SIMULINK R2020a
   V0.04    14.05.2020    Schmidt,   B&R blocks upgrade to AS Target v6.2.0 (officially supports MATLAB 2020a)
   V0.05    03.08.2020    Schmidt,   changed speed reference for function activation from nominal speed (parameter) to bus bar frequency
   added detection for speed exceedance --> switch over to standard idle controller
   V0.06    04.08.2020    Schmidt,   moved function activation from PARA bus to IN bus
   V0.07    17.08.2020    Schmidt,   included modifications after P6 tests
   V0.08    25.01.2021    Schmidt,   use of frequency based speed set-point (rN_Set) only if rF_MMD_BusBar > 0.5*rF_Nom
 ********************************************************************
 * Implementation of program FSyPrM
 ********************************************************************
 * Generated with B&R Automation Studio Target for Simulink V6.3.1
 * (ERT based)
 ********************************************************************/

#include <bur/plctypes.h>
#include "FSyPrM.h"
#include "rtwtypes.h"

/* Defines */
#define SS_TERMINATE 4
#define SS_OUTPUT 3
#define SS_INITIALIZE 2

/*  Data Types */

/**************************** GLOBAL DATA *************************************/
/*  Definitions */

/*  Declarations  */

/***************************** FILE SCOPE DATA ********************************/

/*************************** FUNCTIONS ****************************************/
#ifdef __cplusplus

unsigned long bur_heap_size = 6553500;

#endif

/*LEGACYMODE_VARIABLES*/
void fFSyPrM(struct fFSyPrM* inst)
{
  tag_RTM_FSyPrM* const FSyPrM_M = &(inst)->bur_FSyPrM;
	inst->bur_FSyPrM.blockIO = &(inst)->bur_BlockIO_FSyPrM;
	inst->bur_FSyPrM.inputs = &(inst)->bur_ExternalInputs_FSyPrM;
	inst->bur_FSyPrM.outputs = &(inst)->bur_ExternalOutputs_FSyPrM;
	inst->bur_FSyPrM.dwork = &(inst)->bur_D_Work_FSyPrM;

  switch (inst->ssMethodType)
  {
   case SS_INITIALIZE:
    /* call model initialize function */
    FSyPrM_initialize(FSyPrM_M, inst);
    break;

   case SS_OUTPUT:
    /* call model step function */
    FSyPrM_step(FSyPrM_M, inst);

    break;

   case SS_TERMINATE:
    /* call model terminate function */
    FSyPrM_terminate(FSyPrM_M, inst);
    break;
  }
}

/*****************************************************************************
   Function block sample time: 0.01s
 *****************************************************************************/

/*****************************************************************************
   B&R Automation Studio Target for Simulink Version: A6.3.1 (15-Dec-2020)
 *****************************************************************************/

/*======================== TOOL VERSION INFORMATION ==========================*
 * MATLAB 9.8 (R2020a)18-Nov-2019                                             *
 * Simulink 10.1 (R2020a)18-Nov-2019                                          *
 * Simulink Coder 9.3 (R2020a)18-Nov-2019                                     *
 * Embedded Coder 7.4 (R2020a)18-Nov-2019                                     *
 * Stateflow 10.2 (R2020a)18-Nov-2019                                         *
 *============================================================================*/

/*======================= LICENSE IN USE INFORMATION =========================*
 * matlab                                                                     *
 * matlab_coder                                                               *
 * real-time_workshop                                                         *
 * rtw_embedded_coder                                                         *
 * simulink                                                                   *
 *============================================================================*/
```

#### lFSyPrM.fun
```iecst
FUNCTION_BLOCK fFSyPrM
  VAR_INPUT
    ssMethodType: SINT;
  END_VAR
  VAR_INPUT
        In : tFSyPrM_IN; (*Inputs to FastSync controller*)
  END_VAR
  VAR_INPUT
        Para : tFSyPrM_PARA; (*Parameters to FastSync controller*)
  END_VAR
  VAR_INPUT
        Perm : tFSyPrM_PERM; (*Perm to FastSync controller*)
  END_VAR
  VAR_OUTPUT
        Dbg : tFSyPrM_DBG; (*Debug from FastSync controller*)
  END_VAR
  VAR_OUTPUT
        bEnabled : BOOL := 0; (*True: Autocode active, False: Switch to standard idle controller*)
  END_VAR
  VAR_OUTPUT
        rRetardITP : REAL := 0; (**)
  END_VAR
  VAR_OUTPUT
        Version : UDINT := 0; (**)
  END_VAR
	VAR
		bur_BlockIO_FSyPrM : BlockIO_FSyPrM;
	END_VAR
	VAR
		bur_ExternalInputs_FSyPrM : ExternalInputs_FSyPrM;
	END_VAR
	VAR
		bur_ExternalOutputs_FSyPrM : ExternalOutputs_FSyPrM;
	END_VAR
	VAR
		bur_D_Work_FSyPrM : D_Work_FSyPrM;
	END_VAR
	VAR
		bur_FSyPrM : tag_RTM_FSyPrM;
	END_VAR
END_FUNCTION_BLOCK
```

#### lFSyPrM.typ
```iecst
TYPE
	tFSyPrM_DBG :  STRUCT
		iRetardCounter :  UINT; (* (-)*)
		rSwitchSurf :  REAL; (* (-)*)
		Sf1 :  BOOL; (* (-)*)
		Sf2 :  BOOL; (* (-)*)
		H3 :  BOOL; (* (-)*)
		H4 :  BOOL; (* (-)*)
		rSmodSlid :  REAL; (* (-)*)
		iCounterSwitch :  UINT; (* (-)*)
		bEna :  BOOL; (* (-)*)
		iCtrSel :  SINT; (* (-)*)
		rN_Set :  REAL; (*Speed set point (rpm)*)
		rN_Eng :  REAL; (*Actual speed (rpm)*)
		bSpdSettled :  BOOL; (* (-)*)
		rN_dot :  REAL; (*Engine speed derivative (rpm/s)*)
	END_STRUCT;

	tFSyPrM_IN :  STRUCT
		bGCB_ON :  BOOL; (*Generator circuit breaker closed (-)*)
		rN_Eng :  REAL; (*Engine speed (rpm)*)
		rF_MMD :  REAL; (*Generator frequency (Hz)*)
		rF_MMD_BusBar :  REAL; (*Bus bar frequency (Hz)*)
		rAng_MMD_Diff :  REAL; (*Electric angle (deg)*)
		bFastSync :  BOOL; (*Fast synchronization activation (-)*)
		bReset :  BOOL; (*Reset library (-)*)
	END_STRUCT;

	tFSyPrM_PARA :  STRUCT
		rF_Nom :  REAL; (*Nominal generator frequency (Hz)*)
		rN_EngNom :  REAL; (*Nominal engine speed (rpm)*)
	END_STRUCT;

	tFSyPrM_PERM :  STRUCT
		bSpeedSet_ena :  BOOL; (*Select the setpoint (1: constant speed, 0: grid frequency) (-)*)
		iCtrSel :  SINT; (*Control selection. 1-Std skip firing, 2-Time optimal, 3-Time optimal with constraints, 4-Fuel and time optimal (-)*)
		rAngleSetDeg :  REAL; (*Electric angle setpoint (deg)*)
		rRelaxAngleDeg :  REAL; (*Relaxation band for the electric angle setpoint (deg)*)
		rWeightFuel :  REAL; (*Weighting (high->time, low->fuel) (-)*)
		rHystOptimal :  REAL; (*Band around switching surface (nonnegative >=0) (-)*)
		rCA_ITPRetardMax :  REAL; (*Maximum ITP retard angle (<=20) (CAD)*)
		rCA_ITPRetardMin :  REAL; (*Minimum ITP retard angle (>=0) (CAD)*)
		rTi_FiltF :  REAL; (*Filter constant for grid frequency (s)*)
		rTi_Filtn :  REAL; (*Filter constant for engine speed (s)*)
		rN_enableNorm :  REAL; (*Engine speed normalized to enable fast sync controller (-)*)
		rN_dot_release :  REAL; (*Engine speed derivation threshold (-)*)
		rN_SpdSettled :  REAL; (*Engine speed activation threshold (rpm)*)
		rN_SpdDevMax :  REAL; (*Maximum allowed speed deviation (rpm)*)
		rTi_FastSync :  REAL; (*Switch over to standard controller after this time (s)*)
		bF_act_ena :  BOOL; (*Use generator frequency as actual value (-)*)
	END_STRUCT;

END_TYPE

TYPE
BlockIO_FSyPrM : STRUCT
	BusInput2 : tFSyPrM_PERM;
	BusInput : tFSyPrM_IN;
	BusInput1 : tFSyPrM_PARA;
	UnitDelay : UDINT;
	bEnabled : BOOL;
END_STRUCT;
D_Work_FSyPrM : STRUCT
	DiscreteTimeIntegrator_DSTATE : REAL;
	DiscreteTimeIntegrator_DSTATE_g : REAL;
	DiscreteTimeIntegrator_DSTATE_k : REAL;
	UnitDelay_DSTATE : UDINT;
	CA_retarded : REAL;
	retardcounter : UINT;
	Count_Switch : UINT;
	DiscreteTimeIntegrator_PrevRese : SINT;
	DiscreteTimeIntegrator_PrevRe_h : SINT;
	DiscreteTimeIntegrator_PrevRe_d : SINT;
	DiscreteTimeIntegrator_IC_LOADI : USINT;
	DiscreteTimeIntegrator_IC_LOA_d : USINT;
	DiscreteTimeIntegrator_IC_LO_dn : USINT;
	ssr : BOOL;
	spd_DevExc : BOOL;
	spd_settled : BOOL;
	CA_retarded_not_empty : BOOL;
END_STRUCT;
ExternalInputs_FSyPrM : STRUCT
	In : tFSyPrM_IN;
	Para : tFSyPrM_PARA;
	Perm : tFSyPrM_PERM;
END_STRUCT;
ExternalOutputs_FSyPrM : STRUCT
	rRetardITP : REAL;
	dbg : tFSyPrM_DBG;
END_STRUCT;
tag_RTM_FSyPrM : STRUCT
	errorStatus : REFERENCE TO USINT;
	blockIO : REFERENCE TO BlockIO_FSyPrM;
	inputs : REFERENCE TO ExternalInputs_FSyPrM;
	outputs : REFERENCE TO ExternalOutputs_FSyPrM;
	dwork : REFERENCE TO D_Work_FSyPrM;
END_STRUCT;
RT_MODEL_FSyPrM : tag_RTM_FSyPrM;

END_TYPE
TYPE
END_TYPE
```

#### lib_properties.txt
```
For manual assignment to hardware configuration please
add the following additional include directories:

\Logical\MATLAB_includes\R2020a\

And the following additional build options:

-lm -D MODEL=FSyPrM -D NUMST=1 -D NCSTATES=0 -D HAVESTDIO -D MODEL_HAS_DYNAMICALLY_LOADED_SFCNS=0 -D CLASSIC_INTERFACE=0 -D ALLOCATIONFCN=0 -D TID01EQ=0 -D TERMFCN=1 -D ONESTEPFCN=1 -D MAT_FILE=0 -D MULTI_INSTANCE_CODE=1 -D INTEGER_CODE=0 -D MT=0
```

#### rt_defines.h
```c
/********************************************************************
 * COPYRIGHT -- B&R Industrial Automation GmbH
 ********************************************************************
 * Program: FSyPrM
 * File: rt_defines.h
 * Author: 105055527
 * Last modified by: schmisi00
 * Created: Mon Sep 05 18:14:57 2016
 * Last modified: Mon Jan 25 17:32:20 2021
 * Model Version: 0.08
 * Description: Fast synchronization controller for pre-mixed engines.

   Outstandings:
   -------------
   - NA
 * modified Comment: V0.01    30.03.2020    Schmidt,   project/controller carryover from FSync to FSyncPrM
   V0.02    02.04.2020    Schmidt,   cleanup and deletion of functions not used by pre-mixed engines
   V0.03    12.05.2020    Schmidt,   upgrade to MATLAB/SIMULINK R2020a
   V0.04    14.05.2020    Schmidt,   B&R blocks upgrade to AS Target v6.2.0 (officially supports MATLAB 2020a)
   V0.05    03.08.2020    Schmidt,   changed speed reference for function activation from nominal speed (parameter) to bus bar frequency
   added detection for speed exceedance --> switch over to standard idle controller
   V0.06    04.08.2020    Schmidt,   moved function activation from PARA bus to IN bus
   V0.07    17.08.2020    Schmidt,   included modifications after P6 tests
   V0.08    25.01.2021    Schmidt,   use of frequency based speed set-point (rN_Set) only if rF_MMD_BusBar > 0.5*rF_Nom
 ********************************************************************
 * Header for program FSyPrM
 ********************************************************************
 * Generated with B&R Automation Studio Target for Simulink V6.3.1
 * (ERT based)
 ********************************************************************/

#ifndef RTW_HEADER_rt_defines_h_
#define RTW_HEADER_rt_defines_h_
#ifndef MIN
#define MIN(a,b)                       ((a) < (b) ? (a) : (b))
#endif

#ifndef MAX
#define MAX(a,b)                       ((a) > (b) ? (a) : (b))
#endif

#ifndef AST_ROUND
#define AST_ROUND(x)                   ((x)>=0?(long long)((x)+0.5):(long long)((x)-0.5))
#endif

/*===========*
 * Constants *
 *===========*/
#define RT_PI                          3.14159265358979323846
#define RT_PIF                         3.1415927F
#define RT_LN_10                       2.30258509299404568402
#define RT_LN_10F                      2.3025851F
#define RT_LOG10E                      0.43429448190325182765
#define RT_LOG10EF                     0.43429449F
#define RT_E                           2.7182818284590452354
#define RT_EF                          2.7182817F

/*
 * UNUSED_PARAMETER(x)
 *   Used to specify that a function parameter (argument) is required but not
 *   accessed by the function body.
 */
#ifndef UNUSED_PARAMETER
# if defined(__LCC__)
#   define UNUSED_PARAMETER(x)                                   /* do nothing */
# else

/*
 * This is the semi-ANSI standard way of indicating that an
 * unused function parameter is required.
 */
#   define UNUSED_PARAMETER(x)         (void) (x)
# endif
#endif
#endif                                 /* RTW_HEADER_rt_defines_h_ */
```

#### rtwtypes.h
```c
/********************************************************************
 * COPYRIGHT -- B&R Industrial Automation GmbH
 ********************************************************************
 * Program: FSyPrM
 * File: rtwtypes.h
 * Author: 105055527
 * Last modified by: schmisi00
 * Created: Mon Sep 05 18:14:57 2016
 * Last modified: Mon Jan 25 17:32:20 2021
 * Model Version: 0.08
 * Description: Fast synchronization controller for pre-mixed engines.

   Outstandings:
   -------------
   - NA
 * modified Comment: V0.01    30.03.2020    Schmidt,   project/controller carryover from FSync to FSyncPrM
   V0.02    02.04.2020    Schmidt,   cleanup and deletion of functions not used by pre-mixed engines
   V0.03    12.05.2020    Schmidt,   upgrade to MATLAB/SIMULINK R2020a
   V0.04    14.05.2020    Schmidt,   B&R blocks upgrade to AS Target v6.2.0 (officially supports MATLAB 2020a)
   V0.05    03.08.2020    Schmidt,   changed speed reference for function activation from nominal speed (parameter) to bus bar frequency
   added detection for speed exceedance --> switch over to standard idle controller
   V0.06    04.08.2020    Schmidt,   moved function activation from PARA bus to IN bus
   V0.07    17.08.2020    Schmidt,   included modifications after P6 tests
   V0.08    25.01.2021    Schmidt,   use of frequency based speed set-point (rN_Set) only if rF_MMD_BusBar > 0.5*rF_Nom
 ********************************************************************
 * Header for program FSyPrM
 ********************************************************************
 * Generated with B&R Automation Studio Target for Simulink V6.3.1
 * (ERT based)
 ********************************************************************/

#ifndef RTWTYPES_H
#define RTWTYPES_H

/* Logical type definitions */
#if (!defined(__cplusplus))
#  ifndef false
#   define false                       (0U)
#  endif

#  ifndef true
#   define true                        (1U)
#  endif
#endif

/*=======================================================================*
 * Target hardware information
 *   Device type: Intel->x86/Pentium
 *   Number of bits:     char:   8    short:   16    long:  32
 *                       long:  32
 *                       native word size:  32
 *   Byte ordering: LittleEndian
 *   Signed integer division rounds to: Zero
 *   Shift right on a signed integer as arithmetic shift: on
 *=======================================================================*/

/*=======================================================================*
 * Fixed width word size data types:                                     *
 *   int8_T, int16_T, int32_T     - signed 8, 16, or 32 bit integers     *
 *   uint8_T, uint16_T, uint32_T  - unsigned 8, 16, or 32 bit integers   *
 *   real32_T, real64_T           - 32 and 64 bit floating point numbers *
 *=======================================================================*/
typedef signed char int8_T;
typedef unsigned char uint8_T;
typedef short int16_T;
typedef unsigned short uint16_T;
typedef long int32_T;
typedef unsigned long uint32_T;
typedef float real32_T;
typedef double real64_T;

/*===========================================================================*
 * Generic type definitions: boolean_T, char_T, byte_T, int_T, uint_T,       *
 *                           real_T, time_T, ulong_T.                        *
 *===========================================================================*/
typedef double real_T;
typedef double time_T;
typedef unsigned char boolean_T;
typedef long int_T;
typedef unsigned long uint_T;
typedef unsigned long ulong_T;
typedef char char_T;
typedef unsigned char uchar_T;
typedef char_T byte_T;

/*=======================================================================*
 * Min and Max:                                                          *
 *   int8_T, int16_T, int32_T     - signed 8, 16, or 32 bit integers     *
 *   uint8_T, uint16_T, uint32_T  - unsigned 8, 16, or 32 bit integers   *
 *=======================================================================*/
#define MAX_int8_T                     ((int8_T)(127))
#define MIN_int8_T                     ((int8_T)(-128))
#define MAX_uint8_T                    ((uint8_T)(255U))
#define MAX_int16_T                    ((int16_T)(32767))
#define MIN_int16_T                    ((int16_T)(-32768))
#define MAX_uint16_T                   ((uint16_T)(65535U))
#define MAX_int32_T                    ((int32_T)(2147483647))
#define MIN_int32_T                    ((int32_T)(-2147483647-1))
#define MAX_uint32_T                   ((uint32_T)(0xFFFFFFFFU))

/* Block D-Work pointer type */
typedef void * pointer_T;

#endif                                 /* RTWTYPES_H */

#ifndef MIN
#define MIN(a,b)                       ((a) < (b) ? (a) : (b))
#endif

#ifndef MAX
#define MAX(a,b)                       ((a) > (b) ? (a) : (b))
#endif

#ifndef AST_ROUND
#define AST_ROUND(x)                   ((x)>=0?(long long)((x)+0.5):(long long)((x)-0.5))
#endif
```

### Library Logical/EngineController/Lib_EC/lLamCtrPBC (ANSIC, version 0.00.2)

#### LamCtrPBC.c
```c
/********************************************************************
 * COPYRIGHT -- B&R Industrial Automation GmbH
 ********************************************************************
 * Program: LamCtrPBC
 * File: LamCtrPBC.c
 * Author: kafkama00
 * Last modified by: kafkama00
 * Created: Mon Oct 11 17:08:29 2021
 * Last modified: Wed Dec 01 09:46:51 2021
 * Model Version: 1.00
 * Description: Lambda controller for pressure based control engines
 * modified Comment: V0.01 11.10.2021 created for first tests
   V0.02 12.10.2021 added debug signals
   V0.03 17.11.2021 added distortion rejection
   V1.00 01.12.2021 remove distortion rejection, serial release DIA.NE V4.11
 ********************************************************************
 * Implementation of program LamCtrPBC
 ********************************************************************
 * Generated with B&R Automation Studio Target for Simulink V6.4.1
 * (ERT based)
 ********************************************************************/

#include "LamCtrPBC.h"
#include "LamCtrPBC_private.h"

/*  Defines */

/*  Data Types */

/**************************** GLOBAL DATA *************************************/
/*  Definitions */
const LamCtrPBC_OUT_Bus LamCtrPBC_rtZLamCtrPBC_OUT_Bus = {
  0.0F                                 /* rLam_ref */
} ;                                    /* LamCtrPBC_OUT_Bus ground */

const LamCtrPBC_DBG_Bus LamCtrPBC_rtZLamCtrPBC_DBG_Bus = {
  0.0F,                                /* e_lam */
  0.0F,                                /* u */
  0.0F,                                /* u_lim */
  0.0F,                                /* up_LamCtr */
  0.0F,                                /* ui_LamCtr */
  0.0F,                                /* uAW_LamCtr */
  0.0F,                                /* u_PT1_smith */
  0.0F,                                /* u_delay_smith */
  0.0F                                 /* fb_smith */
} ;                                    /* LamCtrPBC_DBG_Bus ground */

/*  Declarations  */
const LamCtrPBC_IN_Bus LamCtrPBC_rtZLamCtrPBC_IN_Bus = { 0.0F,/* rLam_Set */
  0.0F,                                /* rLam_PBC */
  false                                /* bReset */
};

const LamCtrPBC_PARA_Bus LamCtrPBC_rtZLamCtrPBC_PARA_Bus = { 0.0F,/* rKp_LamCtr */
  0.0F,                                /* rKi_LamCtr */
  0.0F,                                /* rKAW_LamCtr */
  0.0F,                                /* rulim_LamCtr_up */
  0.0F                                 /* rulim_LamCtr_low */
};

const LamCtrPBC_PERM_Bus LamCtrPBC_rtZLamCtrPBC_PERM_Bus = { 0,/* iTd_smith_LamCtr */
  0.0F                                 /* rTi_smith_LamCtr */
};

/***************************** FILE SCOPE DATA ********************************/

/*************************** FUNCTIONS ****************************************/

/* Model step function */
void LamCtrPBC_step(RT_MODEL_LamCtrPBC *const LamCtrPBC_M, struct fLamCtrPBC* inst)
{
  struct BlockIO_LamCtrPBC *LamCtrPBC_B = ((struct BlockIO_LamCtrPBC *) LamCtrPBC_M->blockIO);
  struct D_Work_LamCtrPBC *LamCtrPBC_DWork = ((struct D_Work_LamCtrPBC *) LamCtrPBC_M->dwork);
  struct PrevZCSigStates_LamCtrPBC *LamCtrPBC_PrevZCSigState =
    ((struct PrevZCSigStates_LamCtrPBC *) LamCtrPBC_M->prevZCSigState);
  ExternalOutputs_LamCtrPBC *LamCtrPBC_Y = (ExternalOutputs_LamCtrPBC *)
    LamCtrPBC_M->outputs;
  real32_T rtb_e_lam;
  real32_T rtb_u_delay_smith;
  real32_T rtb_up_LamCtr;
  real32_T rtb_uAW_LamCtr;
  real32_T rtb_u;
  boolean_T rtb_RelationalOperator;
  real32_T rtb_Switch2;
  real32_T rtb_Switch_p;
  real32_T rtb_Switch1;
  real32_T rtb_rLam_ref;
  real32_T rtb_EnvironmentSwitch_o_rLam_PB;
  boolean_T rtb_EnvironmentSwitch_o_bReset;
  real32_T rtb_EnvironmentSwitch_rKi_LamCt;
  boolean_T rtb_LogicalOperator;
  int32_T i;
  int8_T tmp;

  /* S-Function (bur_bus_in): '<Root>/Bus Input' */
  LamCtrPBC_B->BusInput = inst->In;

  /* Switch: '<S1>/Environment Switch' */
  rtb_EnvironmentSwitch_o_rLam_PB = LamCtrPBC_B->BusInput.rLam_PBC;
  rtb_EnvironmentSwitch_o_bReset = LamCtrPBC_B->BusInput.bReset;

  /* Delay: '<Root>/Delay1' incorporates:
   *  DiscreteIntegrator: '<Root>/Discrete-Time Integrator'
   *  Switch: '<S1>/Environment Switch'
   */
  rtb_RelationalOperator = !LamCtrPBC_B->BusInput.bReset;
  if (rtb_RelationalOperator && (LamCtrPBC_PrevZCSigState->Delay1_Reset_ZCE !=
       ZERO_ZCSIG)) {
    LamCtrPBC_DWork->icLoad = 1U;
  }

  LamCtrPBC_PrevZCSigState->Delay1_Reset_ZCE = LamCtrPBC_B->BusInput.bReset;
  if (LamCtrPBC_DWork->icLoad != 0) {
    LamCtrPBC_DWork->Delay1_DSTATE = LamCtrPBC_B->BusInput.rLam_Set;
  }

  /* Sum: '<Root>/Sum' incorporates:
   *  Delay: '<Root>/Delay1'
   *  Switch: '<S1>/Environment Switch'
   */
  rtb_e_lam = LamCtrPBC_B->BusInput.rLam_Set - LamCtrPBC_DWork->Delay1_DSTATE;

  /* S-Function (bur_bus_in): '<Root>/Bus Input1' */
  LamCtrPBC_B->BusInput1 = inst->Para;

  /* Switch: '<S2>/Environment Switch' */
  rtb_EnvironmentSwitch_rKi_LamCt = LamCtrPBC_B->BusInput1.rKi_LamCtr;

  /* Product: '<Root>/Product' incorporates:
   *  Switch: '<S2>/Environment Switch'
   */
  rtb_up_LamCtr = LamCtrPBC_B->BusInput1.rKp_LamCtr * rtb_e_lam;

  /* DiscreteIntegrator: '<Root>/Discrete-Time Integrator' */
  if (rtb_RelationalOperator &&
      (LamCtrPBC_DWork->DiscreteTimeIntegrator_PrevRese == 1)) {
    LamCtrPBC_DWork->DiscreteTimeIntegrator_DSTATE = 0.0F;
  }

  /* Sum: '<Root>/Sum2' incorporates:
   *  DiscreteIntegrator: '<Root>/Discrete-Time Integrator'
   */
  rtb_u = rtb_up_LamCtr + LamCtrPBC_DWork->DiscreteTimeIntegrator_DSTATE;

  /* Switch: '<S6>/Switch2' incorporates:
   *  RelationalOperator: '<S6>/LowerRelop1'
   *  RelationalOperator: '<S6>/UpperRelop'
   *  Switch: '<S2>/Environment Switch'
   *  Switch: '<S6>/Switch'
   */
  if (rtb_u > LamCtrPBC_B->BusInput1.rulim_LamCtr_up) {
    rtb_Switch2 = LamCtrPBC_B->BusInput1.rulim_LamCtr_up;
  } else if (rtb_u < LamCtrPBC_B->BusInput1.rulim_LamCtr_low) {
    /* Switch: '<S6>/Switch' */
    rtb_Switch2 = LamCtrPBC_B->BusInput1.rulim_LamCtr_low;
  } else {
    rtb_Switch2 = rtb_u;
  }

  /* End of Switch: '<S6>/Switch2' */

  /* Product: '<Root>/Product2' incorporates:
   *  Sum: '<Root>/Sum5'
   *  Switch: '<S2>/Environment Switch'
   */
  rtb_uAW_LamCtr = (rtb_u - rtb_Switch2) * LamCtrPBC_B->BusInput1.rKAW_LamCtr;

  /* Switch: '<Root>/Switch' incorporates:
   *  Sum: '<Root>/Sum3'
   *  Switch: '<S1>/Environment Switch'
   */
  if (LamCtrPBC_B->BusInput.bReset) {
    rtb_rLam_ref = LamCtrPBC_B->BusInput.rLam_Set;
  } else {
    rtb_rLam_ref = LamCtrPBC_B->BusInput.rLam_Set + rtb_Switch2;
  }

  /* End of Switch: '<Root>/Switch' */

  /* S-Function (bur_bus_in): '<Root>/Bus Input2' */
  LamCtrPBC_B->BusInput2 = inst->Perm;

  /* Outputs for Atomic SubSystem: '<Root>/Filter2' */
  /* RelationalOperator: '<S4>/Relational Operator' incorporates:
   *  Constant: '<S4>/Constant'
   *  Switch: '<S3>/Environment Switch'
   */
  rtb_RelationalOperator = (LamCtrPBC_B->BusInput2.rTi_smith_LamCtr > 0.0F);

  /* Logic: '<S4>/Logical Operator' incorporates:
   *  Logic: '<S4>/Logical Operator1'
   *  Switch: '<S1>/Environment Switch'
   */
  rtb_LogicalOperator = (LamCtrPBC_B->BusInput.bReset ||
    (!rtb_RelationalOperator));

  /* DiscreteIntegrator: '<S4>/Discrete-Time Integrator' */
  if (LamCtrPBC_DWork->DiscreteTimeIntegrator_IC_LOADI != 0) {
    LamCtrPBC_DWork->DiscreteTimeIntegrator_DSTATE_n = rtb_rLam_ref;
  }

  if (rtb_LogicalOperator || (LamCtrPBC_DWork->DiscreteTimeIntegrator_PrevRe_m
       != 0)) {
    LamCtrPBC_DWork->DiscreteTimeIntegrator_DSTATE_n = rtb_rLam_ref;
  }

  /* Switch: '<S4>/Switch' incorporates:
   *  DiscreteIntegrator: '<S4>/Discrete-Time Integrator'
   */
  if (rtb_RelationalOperator) {
    rtb_Switch_p = LamCtrPBC_DWork->DiscreteTimeIntegrator_DSTATE_n;
  } else {
    rtb_Switch_p = rtb_rLam_ref;
  }

  /* End of Switch: '<S4>/Switch' */

  /* Update for DiscreteIntegrator: '<S4>/Discrete-Time Integrator' */
  LamCtrPBC_DWork->DiscreteTimeIntegrator_IC_LOADI = 0U;

  /* Switch: '<S7>/Switch' incorporates:
   *  Abs: '<S7>/Abs'
   *  RelationalOperator: '<S7>/Relational Operator'
   *  Switch: '<S3>/Environment Switch'
   */
  if (LamCtrPBC_ConstB.Conversion >= fabsf
      (LamCtrPBC_B->BusInput2.rTi_smith_LamCtr)) {
    rtb_u_delay_smith = LamCtrPBC_ConstB.Conversion;
  } else {
    rtb_u_delay_smith = LamCtrPBC_B->BusInput2.rTi_smith_LamCtr;
  }

  /* End of Switch: '<S7>/Switch' */

  /* Update for DiscreteIntegrator: '<S4>/Discrete-Time Integrator' incorporates:
   *  Product: '<S4>/Divide4'
   *  Sum: '<S4>/Sum4'
   */
  LamCtrPBC_DWork->DiscreteTimeIntegrator_DSTATE_n += (rtb_rLam_ref -
    LamCtrPBC_DWork->DiscreteTimeIntegrator_DSTATE_n) / rtb_u_delay_smith *
    0.01F;
  LamCtrPBC_DWork->DiscreteTimeIntegrator_PrevRe_m = (int8_T)rtb_LogicalOperator;

  /* End of Outputs for SubSystem: '<Root>/Filter2' */

  /* Delay: '<Root>/Delay' incorporates:
   *  Switch: '<S3>/Environment Switch'
   */
  if (LamCtrPBC_DWork->icLoad_o != 0) {
    for (i = 0; i < 50; i++) {
      LamCtrPBC_DWork->Delay_DSTATE[i] = rtb_Switch_p;
    }
  }

  if (LamCtrPBC_B->BusInput2.iTd_smith_LamCtr <= 0) {
    rtb_u_delay_smith = rtb_Switch_p;
  } else {
    if (LamCtrPBC_B->BusInput2.iTd_smith_LamCtr > 50) {
      tmp = 50;
    } else {
      tmp = LamCtrPBC_B->BusInput2.iTd_smith_LamCtr;
    }

    rtb_u_delay_smith = LamCtrPBC_DWork->Delay_DSTATE[(int8_T)(50 - tmp)];
  }

  /* End of Delay: '<Root>/Delay' */

  /* Sum: '<Root>/Sum6' */
  rtb_Switch1 = rtb_Switch_p - rtb_u_delay_smith;

  /* Outport: '<Root>/dbg' incorporates:
   *  BusCreator generated from: '<Root>/dbg'
   *  DiscreteIntegrator: '<Root>/Discrete-Time Integrator'
   */
  LamCtrPBC_Y->dbg.e_lam = rtb_e_lam;
  LamCtrPBC_Y->dbg.u = rtb_u;
  LamCtrPBC_Y->dbg.u_lim = rtb_Switch2;
  LamCtrPBC_Y->dbg.up_LamCtr = rtb_up_LamCtr;
  LamCtrPBC_Y->dbg.ui_LamCtr = LamCtrPBC_DWork->DiscreteTimeIntegrator_DSTATE;
  LamCtrPBC_Y->dbg.uAW_LamCtr = rtb_uAW_LamCtr;
  LamCtrPBC_Y->dbg.u_PT1_smith = rtb_Switch_p;
  LamCtrPBC_Y->dbg.u_delay_smith = rtb_u_delay_smith;
  LamCtrPBC_Y->dbg.fb_smith = rtb_Switch1;

  /* BusCreator generated from: '<Root>/Bus Output1' incorporates:
   *  DiscreteIntegrator: '<Root>/Discrete-Time Integrator'
   */
  LamCtrPBC_B->BusConversion_InsertedFor_BusOu.e_lam = rtb_e_lam;
  LamCtrPBC_B->BusConversion_InsertedFor_BusOu.u = rtb_u;
  LamCtrPBC_B->BusConversion_InsertedFor_BusOu.u_lim = rtb_Switch2;
  LamCtrPBC_B->BusConversion_InsertedFor_BusOu.up_LamCtr = rtb_up_LamCtr;
  LamCtrPBC_B->BusConversion_InsertedFor_BusOu.ui_LamCtr =
    LamCtrPBC_DWork->DiscreteTimeIntegrator_DSTATE;
  LamCtrPBC_B->BusConversion_InsertedFor_BusOu.uAW_LamCtr = rtb_uAW_LamCtr;
  LamCtrPBC_B->BusConversion_InsertedFor_BusOu.u_PT1_smith = rtb_Switch_p;
  LamCtrPBC_B->BusConversion_InsertedFor_BusOu.u_delay_smith = rtb_u_delay_smith;
  LamCtrPBC_B->BusConversion_InsertedFor_BusOu.fb_smith = rtb_Switch1;

  /* BusCreator generated from: '<Root>/Bus Output' */
  LamCtrPBC_B->BusConversion_InsertedFor_Bus_b.rLam_ref = rtb_rLam_ref;

  /* S-Function (bur_bus_out): '<Root>/Bus Output' */
  inst->Out = LamCtrPBC_B->BusConversion_InsertedFor_Bus_b;

  /* S-Function (bur_bus_out): '<Root>/Bus Output1' */
  inst->dbg = LamCtrPBC_B->BusConversion_InsertedFor_BusOu;

  /* UnitDelay: '<S5>/Unit Delay' */
  LamCtrPBC_B->UnitDelay = LamCtrPBC_DWork->UnitDelay_DSTATE;

  /* S-Function (bur_out): '<Root>/Output' */
  inst->Version = LamCtrPBC_B->UnitDelay;

  /* Switch: '<Root>/Switch1' incorporates:
   *  Constant: '<Root>/Constant'
   *  Switch: '<S3>/Environment Switch'
   */
  if (LamCtrPBC_B->BusInput2.iTd_smith_LamCtr <= 0) {
    rtb_Switch1 = 0.0F;
  }

  /* End of Switch: '<Root>/Switch1' */

  /* Outport: '<Root>/Out' incorporates:
   *  BusCreator generated from: '<Root>/Out'
   */
  LamCtrPBC_Y->Out.rLam_ref = rtb_rLam_ref;

  /* Update for Delay: '<Root>/Delay1' incorporates:
   *  Sum: '<Root>/Sum1'
   */
  LamCtrPBC_DWork->icLoad = 0U;
  LamCtrPBC_DWork->Delay1_DSTATE = rtb_EnvironmentSwitch_o_rLam_PB + rtb_Switch1;

  /* Update for DiscreteIntegrator: '<Root>/Discrete-Time Integrator' incorporates:
   *  Product: '<Root>/Product1'
   *  Sum: '<Root>/Sum4'
   */
  LamCtrPBC_DWork->DiscreteTimeIntegrator_DSTATE += (rtb_e_lam *
    rtb_EnvironmentSwitch_rKi_LamCt - rtb_uAW_LamCtr) * 0.01F;
  LamCtrPBC_DWork->DiscreteTimeIntegrator_PrevRese = (int8_T)
    rtb_EnvironmentSwitch_o_bReset;

  /* Update for Delay: '<Root>/Delay' */
  LamCtrPBC_DWork->icLoad_o = 0U;
  for (i = 0; i < 49; i++) {
    LamCtrPBC_DWork->Delay_DSTATE[i] = LamCtrPBC_DWork->Delay_DSTATE[i + 1];
  }

  LamCtrPBC_DWork->Delay_DSTATE[49] = rtb_Switch_p;

  /* End of Update for Delay: '<Root>/Delay' */

  /* Update for UnitDelay: '<S5>/Unit Delay' */
  LamCtrPBC_DWork->UnitDelay_DSTATE = LamCtrPBC_ConstB.DataTypeConversion3;
}

/* Model initialize function */
void LamCtrPBC_initialize(RT_MODEL_LamCtrPBC *const LamCtrPBC_M, struct fLamCtrPBC* inst)
{
  struct D_Work_LamCtrPBC *LamCtrPBC_DWork = ((struct D_Work_LamCtrPBC *) LamCtrPBC_M->dwork);
  struct PrevZCSigStates_LamCtrPBC *LamCtrPBC_PrevZCSigState =
    ((struct PrevZCSigStates_LamCtrPBC *) LamCtrPBC_M->prevZCSigState);
  struct BlockIO_LamCtrPBC *LamCtrPBC_B = ((struct BlockIO_LamCtrPBC *) LamCtrPBC_M->blockIO);
  ExternalInputs_LamCtrPBC *LamCtrPBC_U = (ExternalInputs_LamCtrPBC *)
    LamCtrPBC_M->inputs;
  ExternalOutputs_LamCtrPBC *LamCtrPBC_Y = (ExternalOutputs_LamCtrPBC *)
    LamCtrPBC_M->outputs;

  /* Registration code */

  /* block I/O */
  (void) memset(((void *) LamCtrPBC_B), 0,
                sizeof(struct BlockIO_LamCtrPBC));

  {
    LamCtrPBC_B->BusConversion_InsertedFor_BusOu =
      LamCtrPBC_rtZLamCtrPBC_DBG_Bus;
    LamCtrPBC_B->BusInput1 = LamCtrPBC_rtZLamCtrPBC_PARA_Bus;
    LamCtrPBC_B->BusInput = LamCtrPBC_rtZLamCtrPBC_IN_Bus;
    LamCtrPBC_B->BusInput2 = LamCtrPBC_rtZLamCtrPBC_PERM_Bus;
    LamCtrPBC_B->BusConversion_InsertedFor_Bus_b =
      LamCtrPBC_rtZLamCtrPBC_OUT_Bus;
  }

  /* states (dwork) */
  (void) memset((void *)LamCtrPBC_DWork, 0,
                sizeof(struct D_Work_LamCtrPBC));
  LamCtrPBC_DWork->Delay1_DSTATE = 0.0F;
  LamCtrPBC_DWork->DiscreteTimeIntegrator_DSTATE = 0.0F;

  {
    int32_T i;
    for (i = 0; i < 50; i++) {
      LamCtrPBC_DWork->Delay_DSTATE[i] = 0.0F;
    }
  }

  LamCtrPBC_DWork->DiscreteTimeIntegrator_DSTATE_n = 0.0F;

  /* external inputs */
  LamCtrPBC_U->In = LamCtrPBC_rtZLamCtrPBC_IN_Bus;
  LamCtrPBC_U->Para = LamCtrPBC_rtZLamCtrPBC_PARA_Bus;
  LamCtrPBC_U->Perm = LamCtrPBC_rtZLamCtrPBC_PERM_Bus;

  /* external outputs */
  LamCtrPBC_Y->Out = LamCtrPBC_rtZLamCtrPBC_OUT_Bus;
  LamCtrPBC_Y->dbg = LamCtrPBC_rtZLamCtrPBC_DBG_Bus;
  LamCtrPBC_PrevZCSigState->Delay1_Reset_ZCE = ZERO_ZCSIG;

  /* InitializeConditions for Delay: '<Root>/Delay1' */
  LamCtrPBC_DWork->icLoad = 1U;

  /* InitializeConditions for DiscreteIntegrator: '<Root>/Discrete-Time Integrator' */
  LamCtrPBC_DWork->DiscreteTimeIntegrator_PrevRese = 2;

  /* InitializeConditions for Delay: '<Root>/Delay' */
  LamCtrPBC_DWork->icLoad_o = 1U;

  /* SystemInitialize for Atomic SubSystem: '<Root>/Filter2' */
  /* InitializeConditions for DiscreteIntegrator: '<S4>/Discrete-Time Integrator' */
  LamCtrPBC_DWork->DiscreteTimeIntegrator_PrevRe_m = 0;
  LamCtrPBC_DWork->DiscreteTimeIntegrator_IC_LOADI = 1U;

  /* End of SystemInitialize for SubSystem: '<Root>/Filter2' */
}

/* Model terminate function */
void LamCtrPBC_terminate(RT_MODEL_LamCtrPBC *const LamCtrPBC_M, struct fLamCtrPBC* inst)
{
  /* (no terminate code required) */
  UNUSED_PARAMETER(LamCtrPBC_M);
}

/*======================== TOOL VERSION INFORMATION ==========================*
 * MATLAB 9.8 (R2020a)18-Nov-2019                                             *
 * Simulink 10.1 (R2020a)18-Nov-2019                                          *
 * Simulink Coder 9.3 (R2020a)18-Nov-2019                                     *
 * Embedded Coder 7.4 (R2020a)18-Nov-2019                                     *
 * Stateflow 10.2 (R2020a)18-Nov-2019                                         *
 *============================================================================*/

/*======================= LICENSE IN USE INFORMATION =========================*
 * matlab                                                                     *
 * matlab_coder                                                               *
 * real-time_workshop                                                         *
 * rtw_embedded_coder                                                         *
 * simulink                                                                   *
 *============================================================================*/
```
